// ---- POUs/Coolers/FB_SIM_RS_COMM_CRYOTELGT.TcPOU
FUNCTION_BLOCK FB_SIM_RS_COMM_CRYOTELGT EXTENDS FB_SIM_RS_COMM_BASE
VAR_INPUT
END_VAR
VAR_OUTPUT
END_VAR
VAR
	//
	// Status structure for Cryotel GT devices
	//
	// Status attributes that are read from the controller via RS-232
	sVersion:			STRING	:= 'v1.5.3 SIM';
	sMode:				STRING	:= 'GT';
	sSensor:			STRING	:= 'PT-100';
	sCtrlError:			STRING	:= '00000000';
	sCtrlMode:			STRING	:= 'OFF';
	
	lrPowerMeasured:	LREAL	:= 0.0;
	lrPowerCommanded:	LREAL	:= 240.0;
	lrTempColdHead:		LREAL	:= 289.15;	// Room temperature (289.15K = 16.0C) to start with.
	lrTempReject:		LREAL	:= 25.3;	// [C]
	lrTempTarget:		LREAL	:= 0.0;		// Not used
	
	
	fbTimer:		TON;

END_VAR

M_ActivityDo();	// Implement ramps, if any

SUPER^();

METHOD M_ActivityDo
VAR_INPUT
END_VAR
VAR
	lrProgress:	LREAL;
END_VAR
fbTimer();

IF sCtrlMode = 'POWER' THEN
	IF NOT fbTimer.Q	THEN
		lrProgress		:= TIME_TO_LREAL(fbTimer.ET) / TIME_TO_LREAL(fbTimer.PT);
		lrTempColdHead	:= 	289.15 - (289.15 - 80.0) * lrProgress;
	ELSE
		lrTempColdHead	:= 80.0;
	END_IF
END_IF
END_METHOD

METHOD M_GetSimReply : STRING(255)
VAR_INPUT
	{attribute 'OPC.UA.DA' := '0'}
	in_sReceived:	STRING(255);		// String received from a client
END_VAR
VAR
	sReply:	STRING(255);
	sTempStr:	STRING;
	lrVal:	LREAL;
	i:		INT;
    fbFormat   : FB_FormatString;
    sOut       : T_MaxString;
	nCh:	INT := 8;	// Number of channels for models 218 and 224
END_VAR
// Simulated reply has to include the echo of the command.
// For example:
//    command = 'VERSION'
//    reply   = 'VERSION$R$Nv1.5.3$R'

IF FIND (in_sReceived, 'VERSION') = 1 THEN
	sTempStr		:= CONCAT('VERSION$R$N', sVersion);
	M_GetSimReply	:= CONCAT(sTempStr,in_sReplySuffix);
ELSIF FIND (in_sReceived, 'MODE') = 1 THEN
	sTempStr		:= CONCAT('MODE$R$N', sMode);
	M_GetSimReply	:= CONCAT(sTempStr,in_sReplySuffix);
ELSIF FIND (in_sReceived, 'SENSOR') = 1 THEN
	sTempStr		:= CONCAT('SENSOR$R$N', sSensor);
	M_GetSimReply	:= CONCAT(sTempStr,in_sReplySuffix);
ELSIF FIND (in_sReceived, 'PWOUT=') = 1 THEN
	// Example:         'PWOUT=240$R'.
	// Reply should be: 'PWOUT=240$R$N240.00$R'.
	// Get the value from the command, i.e. everything after 'PWOUT='.
	sTempStr			:= MID(in_sReceived, LEN(in_sReceived)-6, 7);	// = '240$R'
	lrPowerCommanded	:= STRING_TO_LREAL(sTempStr);	// = 240.0
	sTempStr			:= CONCAT(in_sReceived, '$N');	// 'PWOUT=240$R' + '$N' = 'PWOUT=240$R$N' 
	M_GetSimReply		:= CONCAT(sTempStr, M_Get_LREAL_TO_STRING(lrPowerCommanded,2));
ELSIF FIND (in_sReceived, 'PWOUT') = 1 THEN
	M_GetSimReply	:= CONCAT('PWOUT$R$N', M_Get_LREAL_TO_STRING(lrPowerCommanded,2));
ELSIF FIND (in_sReceived, 'P') = 1 THEN
	lrPowerMeasured	:= M_GenerateRandom_LREAL(lrPowerCommanded-0.3,0.3);
	M_GetSimReply	:= CONCAT('P$R$N', M_Get_LREAL_TO_STRING(lrPowerMeasured,2));
ELSIF FIND (in_sReceived, 'ERROR') = 1 THEN
	sTempStr		:= CONCAT('ERROR$R$N', sCtrlError);
	M_GetSimReply	:= CONCAT(sTempStr,in_sReplySuffix);
ELSIF FIND (in_sReceived, 'COOLER=POWER') = 1 THEN
	sCtrlMode		:= 'POWER';
	M_GetSimReply	:= CONCAT('COOLER=POWER$R$NPOWER',in_sReplySuffix);
	// Start ramping down the cold head temperature,
	// starting fromroom temperature.
	lrTempColdHead	:= 289.15;	
	fbTimer(IN:=FALSE);
	fbTimer(IN:=TRUE, PT:=T#60S);
ELSIF FIND (in_sReceived, 'COOLER=OFF') = 1 THEN
	fbTimer(IN:=FALSE);	// Stop the temperature ramp.
	sCtrlMode			:= 'OFF';
	M_GetSimReply		:= CONCAT('COOLER=OFF$R$NOFF',in_sReplySuffix);
	lrPowerCommanded	:= 240.0;
	lrPowerMeasured		:= 0.0;
	lrTempColdHead		:= 289.15;
ELSIF FIND (in_sReceived, 'COOLER') = 1 THEN
	sTempStr		:= CONCAT('COOLER$R$N', sCtrlMode);
	M_GetSimReply	:= CONCAT(sTempStr,in_sReplySuffix);
ELSIF FIND (in_sReceived, 'TC') = 1 THEN
	M_GetSimReply	:= CONCAT('TC$R$N', M_Get_LREAL_TO_STRING(lrTempColdHead,2));
ELSIF FIND (in_sReceived, 'TEMP RJ') = 1 THEN
	// Reject temperature [C] !!! should always be close to 
	// the room temperature and slightly above the 
	// cold head temperature [K].
	// So, we have to convert K to C.
	lrTempReject	:= M_GenerateRandom_LREAL(MAX(16.0,lrTempColdHead-273.15),0.1);
	M_GetSimReply	:= CONCAT('TEMP RJ$R$N', M_Get_LREAL_TO_STRING(lrTempReject,2));
ELSE
	// Unknown command.
	// Return '<CR><LF><CR>', i.e. '$R$N$R' in order to complete the reading.
	M_GetSimReply	:= CONCAT('$R$N', in_sReplySuffix);
END_IF
END_METHOD

END_FUNCTION_BLOCK

// ---- POUs/Subsystems/Examples/Evacuation/FB_SIM_MICADO_VALVES.TcPOU
FUNCTION_BLOCK FB_SIM_MICADO_VALVES
VAR_INPUT
END_VAR
VAR_OUTPUT
END_VAR
VAR
	// Output valve control signals
	i_bON_PVV1	AT %I*:	BOOL;
	i_bON_PVV2	AT %I*:	BOOL;
	i_bON_PVV3	AT %I*:	BOOL;
	i_bON_PVV4	AT %I*:	BOOL;
	i_bON_GBV	AT %I*:	BOOL;
	
	
	// Simulation of ON/open feedback signal
	q_bON_PVV1	AT %Q*:	BOOL := FALSE;
	q_bON_PVV2	AT %Q*:	BOOL := FALSE;
	q_bON_PVV3	AT %Q*:	BOOL := FALSE;
	q_bON_PVV4	AT %Q*:	BOOL := FALSE;
	q_bON_GBV	AT %Q*:	BOOL := FALSE;
	
	// Simulation of OFF/closed feedback signal
	q_bOFF_PVV1	AT %Q*:	BOOL := TRUE;
	q_bOFF_PVV2	AT %Q*:	BOOL := TRUE;
	q_bOFF_PVV3	AT %Q*:	BOOL := TRUE;
	q_bOFF_PVV4	AT %Q*:	BOOL := TRUE;
	q_bOFF_GBV	AT %Q*:	BOOL := TRUE;
	

END_VAR

// ON signals are active low
q_bON_PVV1	:= i_bON_PVV1;
q_bON_PVV2	:= i_bON_PVV2;
q_bON_PVV3	:= i_bON_PVV3;
q_bON_PVV4	:= i_bON_PVV4;
q_bON_GBV	:= i_bON_GBV;


// OFF signals are active low
q_bOFF_PVV1	:= NOT i_bON_PVV1;
q_bOFF_PVV2	:= NOT i_bON_PVV2;
q_bOFF_PVV3	:= NOT i_bON_PVV3;
q_bOFF_PVV4	:= NOT i_bON_PVV4;
q_bOFF_GBV	:= NOT i_bON_GBV;

END_FUNCTION_BLOCK

// ---- POUs/Subsystems/Examples/Evacuation/FB_SIM_MICADO_PUMPS.TcPOU
FUNCTION_BLOCK FB_SIM_MICADO_PUMPS
VAR_INPUT
	in_RefPVP:	REFERENCE TO FB_CRYO_PUMP_ECODRY;
	in_RefTMP:	REFERENCE TO FB_CRYO_PUMP_ATH2303M;
	in_Delay:	TIME := T#10S;
END_VAR
VAR_OUTPUT
END_VAR
VAR
	trgStart_PVP:	R_TRIG;
	trgStart_TMP:	R_TRIG;
	trgStop_PVP:	F_TRIG;
	trgStop_TMP:	F_TRIG;
	
	timer_PVP:		TON;
	timer_TMP:		TON;
	
	bON_PVP:		BOOL := FALSE;
	bON_TMP:		BOOL := FALSE;
	
	q_PVP_Running	AT %Q*:	BOOL := TRUE;	// Active low!
	q_TMP_Ready		AT %Q*:	BOOL;
	q_TMP_Speed100	AT %Q*:	BOOL;
	
	ptrTMP_Speed:	POINTER TO DINT;
END_VAR

// Assign pointer to TMP speed.
ptrTMP_Speed	:= ADR(in_RefTMP.stat.nPumpSpeed);

// Get Start signals
trgStart_PVP(CLK:=in_RefPVP.in_bEnable);
trgStart_TMP(CLK:=in_RefTMP.in_bEnable);

// Get Stop signals
trgStop_PVP(CLK:=in_RefPVP.in_bEnable);
trgStop_TMP(CLK:=in_RefTMP.in_bEnable);

// Start timer on Start/Stop events
IF trgStart_PVP.Q THEN
	bON_PVP	:= TRUE;
	timer_PVP(IN:=FALSE);
	timer_PVP(IN:=TRUE, PT:=in_Delay/2);
ELSIF trgStop_PVP.Q THEN
	bON_PVP	:= FALSE;
	timer_PVP(IN:=FALSE);
	timer_PVP(IN:=TRUE, PT:=in_Delay/2);
END_IF

IF trgStart_TMP.Q THEN
	bON_TMP	:= TRUE;
	timer_TMP(IN:=FALSE);
	timer_TMP(IN:=TRUE, PT:=in_Delay);
ELSIF trgStop_TMP.Q THEN
	bON_TMP	:= FALSE;
	timer_TMP(IN:=FALSE);
	timer_TMP(IN:=TRUE, PT:=in_Delay * 2);
END_IF

// Execute timers
timer_PVP();
timer_TMP();

// Set outputs on timer expiry
IF timer_PVP.Q THEN
	// NOTE: PVP feedback is active low.
	IF bON_PVP THEN
		q_PVP_Running	:= FALSE;
	ELSE
		q_PVP_Running	:= TRUE;
	END_IF
END_IF

IF bON_TMP  AND (NOT timer_TMP.Q AND timer_TMP.ET > T#3S) THEN
	// Starting up.
	// Set speed > 100 rpm after 3 sec.
	ptrTMP_Speed^	:= 500;
	q_TMP_Speed100	:= TRUE;
END_IF

IF NOT bON_TMP  AND (NOT timer_TMP.Q AND timer_TMP.ET > T#5S) THEN
	// Stopping the pump.
	// Not ready after 5 sec.
	// However, the pump is still spinning.
	ptrTMP_Speed^	:= 1800;
	q_TMP_Ready		:= FALSE;
END_IF

IF timer_TMP.Q THEN
	IF bON_TMP THEN
		ptrTMP_Speed^	:= 2000;
		q_TMP_Ready	:= TRUE;
	ELSE
		ptrTMP_Speed^	:= 0;
		q_TMP_Ready		:= FALSE;
		q_TMP_Speed100	:= FALSE;
	END_IF
END_IF

END_FUNCTION_BLOCK

// ---- POUs/Subsystems/Examples/LN2_Precooling/FB_CRYO_LN2_PRECOOL.TcPOU
FUNCTION_BLOCK FB_CRYO_LN2_PRECOOL EXTENDS FB_CRYO_GEN_CTRL_BASE
VAR_INPUT
	in_lrTempK:				LREAL;			// Temperature input value [K]
	in_bTempValid:			BOOL := TRUE;	// Temperature Valid flag
	// Two parameters for decision making
	in_lrTempValveOpen:		LREAL := 91.27;		// Open  valve if temperature above this value [K]
	in_lrTempValveClose:	LREAL := 79.148;	// Close valve if temperature below this value [K]
END_VAR
VAR_OUTPUT
END_VAR
VAR
	// Status structure
	{attribute 'OPC.UA.DA' := '1'}
	stat:				T_CRYO_GEN_CTRL_STATUS_BASE;
	
	// LN2 valve
	valve:				FB_CRYO_VALVE_CTRL;
	bEnable_valve:		BOOL := FALSE;	// Valve open when bEnable_valve = TRUE
		

END_VAR

SUPER^();

METHOD M_ActionOffExecute
VAR_INPUT
END_VAR
//
// In this method the Enable flag of the valve is set to FALSE,
// meaning close the valve.
// 
// In the corresponding Activity M_ActivitySwitchingOff(), 
// the completion of the CLOSE/OFF command will be checked.
//
timer(IN:=FALSE);	// Reset Timer - mandatory!

// Close the valve
bEnable_valve	:= FALSE;
END_METHOD

METHOD M_ActionOnExecute
VAR_INPUT
END_VAR
//
// In this method the Enable flag of the valve is set to TRUE,
// meaning open the valve.
// 
// In the corresponding Activity M_ActivitySwitchingOn(), 
// the completion of the OPEN/ON command will be checked.
//
timer(IN:=FALSE);	// Reset Timer - mandatory!

// Close the valve
bEnable_valve	:= TRUE;
END_METHOD

METHOD M_ActivitySwitchingOff : BOOL
VAR_INPUT
END_VAR
//
// Wait for the valve to CLOSE/OFF.
// The valve state is available in its status structure.
// When complete, the method shall return TRUE, otherwise FALSE.


//
// Execute the timer - mandatory.
// Timer expiry is checked in M_ProcessEvents().
//
timer(IN:=TRUE, PT:=UDINT_TO_TIME(in_nTimeout));
	
// If valve is closed, return TRUE, otherwise FALSE.
IF valve.stat.bActOFF THEN
	M_ActivitySwitchingOff := TRUE;
ELSE
	M_ActivitySwitchingOff := FALSE;
END_IF
END_METHOD

METHOD M_ActivitySwitchingOn : BOOL
VAR_INPUT
END_VAR
//
// Wait for the valve to OPEN/ON.
// The valve state is available in its status structure.
// When complete, the method shall return TRUE, otherwise FALSE.


//
// Execute the timer - mandatory.
// Timer expiry is checked in M_ProcessEvents().
//
timer(IN:=TRUE, PT:=UDINT_TO_TIME(in_nTimeout));
	
// If valve is open, return TRUE, otherwise FALSE.
IF valve.stat.bActON THEN
	M_ActivitySwitchingOn := TRUE;
ELSE
	M_ActivitySwitchingOn := FALSE;
END_IF
END_METHOD

METHOD M_Configure
VAR_INPUT
END_VAR
// Configure the system and set the bConfigured flag to TRUE.

(*
	TODO USER: 
	- Set references to extended structures. e.g.
	     statRef REF=stat;
	- Configure the system.
*)

//	MUST be the very first line!!!
statRef REF=stat;

// The system has been configured
bConfigured := TRUE;
END_METHOD

METHOD M_ControlLoop : BOOL
VAR_INPUT
END_VAR
//
// This method implements the logic for controlling the LN2 valve.
// 
// The return value indicates if the valve should be OPEN/TRUE or CLOSED/FALSE
//
	
CASE statRef.nState OF
	E_CRYO_BIN_CTRL_STATE.ACTIVE_SWITCHING_ON,
	E_CRYO_BIN_CTRL_STATE.ACTIVE_ON:
		IF in_bTempValid AND in_lrTempK < in_lrTempValveClose THEN
			// Temperature too low.
			// Close the valve to stop cooling.
			M_ControlLoop	:= FALSE;
		ELSE
			// Keep the valve open
			M_ControlLoop	:= TRUE;
		END_IF

	E_CRYO_BIN_CTRL_STATE.ACTIVE_SWITCHING_OFF,
	E_CRYO_BIN_CTRL_STATE.ACTIVE_OFF:
		IF in_bTempValid AND in_lrTempK > in_lrTempValveOpen THEN
			// Temperature too high.
			// Open the valve to start cooling.
			M_ControlLoop	:= TRUE;
		ELSE
			// Keep the valve closed
			M_ControlLoop	:= FALSE;
		END_IF
ELSE
	// Keep the valve closed
	M_ControlLoop	:= FALSE;
END_CASE
END_METHOD

METHOD M_ExecuteActuators
VAR_INPUT
END_VAR
(*
	TODO USER: Execute all actuators, e.g. valve, heater, etc.
*)

valve(	in_nTimeout	:= 3000, 
		in_bEnable	:= bEnable_valve);
END_METHOD

METHOD M_IsError : BOOL
VAR_INPUT
END_VAR
//
// Check all possible failure conditions.
//
// This includes:
// - Configuration,
// - Validity of temperature reading,
// - Valve failure.
// 
// Return TRUE in case of errors.
// Set error description as well.
//
IF in_lrTempValveClose >= in_lrTempValveOpen THEN
	// The temperatue at which valve opens must be
	// higher than the one at which it closes.
	M_IsError	:= TRUE;
	stat.sError	:= 'ERROR: Wrong temperature limits!';
ELSIF NOT in_bTempValid	THEN
	// Temperature reading invalid.
	M_IsError	:= TRUE;
	stat.sError	:= 'ERROR: Reference temperature invalid!';
ELSIF valve.stat.bError 	THEN
	// Valve has failed.
	M_IsError	:= TRUE;
	stat.sError	:= 'ERROR: Valve failure!';
ELSE
	M_IsError	:= FALSE;
END_IF
END_METHOD

METHOD M_SetStatus
VAR_INPUT
END_VAR
// Execute M_SetStatus() of the base FB
SUPER^.M_SetStatus();


// Correct for LN2 specific labels

CASE statRef.nState OF
	
	E_CRYO_BIN_CTRL_STATE.ACTIVE_OFF:
	statRef.sState	:= 'ACTIVE_VALVE_CLOSED';
	
	E_CRYO_BIN_CTRL_STATE.ACTIVE_ON:
	statRef.sState	:= 'ACTIVE_VALVE_OPEN';
	
	E_CRYO_BIN_CTRL_STATE.ACTIVE_SWITCHING_ON:
	statRef.sState	:= 'OPENING VALVE...';
	
	E_CRYO_BIN_CTRL_STATE.ACTIVE_SWITCHING_OFF:
	statRef.sState	:= 'CLOSING VALVE...';
	
END_CASE
END_METHOD

END_FUNCTION_BLOCK

// ---- POUs/Actuators/FB_CRYO_GEN_CTRL_BASE.TcPOU
// Generic Controller
FUNCTION_BLOCK FB_CRYO_GEN_CTRL_BASE
VAR_INPUT
	in_bEnable:			BOOL := FALSE;	// Controller active while in_bEnable is TRUE
	in_nTimeout:		UDINT := 10000;	// Timeout for switching on/off [ms]. Default 10000.
	(*
		TODO USER: Add all specific input parameters, e.g.
		- Configuration parameters
		- External variables, e.g. temperature, pressure, etc.
	*)
END_VAR
VAR
	(*
		TODO USER: Add all system actuators, variables and I/O signals, e.g.
		
		{attribute 'OPC.UA.DA' := '1'}
		Actuator:	FB_CRYO_BIN_ACT;	// Heater, valve, etc.
	*)
	
	{attribute 'OPC.UA.DA' := '0'}
	statRef:	REFERENCE TO T_CRYO_GEN_CTRL_STATUS_BASE;

	(*
		TODO USER:	Add a 'stat' structure.
					It can be the T_CRYO_GEN_CTRL_STATUS or a struct that EXTENDS T_CRYO_GEN_CTRL_STATUS.
					For example:
						stat:	T_CRYO_BIN_CTRL_STATUS;
	*)
	
	nEvent:		E_CRYO_GEN_CTRL_EVENT := E_CRYO_GEN_CTRL_EVENT.NONE;

	{attribute 'OPC.UA.DA' := '0'}
	timer:		TON;		// Timer for commands
	
	{attribute 'OPC.UA.DA' := '0'}
	trgEnable:	R_TRIG;		// Rising trigger of in_bEnable
	
	// This flag will be set once M_Configure() is executed.
	bConfigured:	BOOL := FALSE;
END_VAR

// Don't do anything until the controller is configured
IF NOT bConfigured THEN
	M_Configure();
	RETURN;
END_IF

// Increment cycle counter
statRef.nCycleCounter := statRef.nCycleCounter + 1;



M_ReadInputs();


M_ExecuteActuators();


M_SetStatus();


M_CheckForEvents();


M_ProcessEvents();

METHOD M_ActionOffExecute
VAR_INPUT
END_VAR
//
// In this method the user shall turn off the actuator(s) such as valves, heaters, coolers, etc.
// Normally this is done by setting the in_bEnable flag of the actuator to FALSE.
// In the corresponding Activity M_ActivitySwitchingOff(), the completion of the OFF command shall be checked.
//
timer(IN:=FALSE);	// Reset Timer - mandatory!
END_METHOD

METHOD M_ActionOnExecute
VAR_INPUT
END_VAR
// In this method the user shall turn on the actuator(s) such as valves, heaters, coolers, etc.
// Normally this is done by setting the in_bEnable flag of the actuator to TRUE.
// In the corresponding Activity M_ActivitySwitchingOn(), the completion of the ON command shall be checked.
timer(IN:=FALSE);	// Reset Timer
END_METHOD

METHOD M_ActivitySwitchingOff : BOOL
VAR_INPUT
END_VAR
// In this method the user shall wait until the actuator is turned OFF.
// The actuator state is available in the status structure.
// When complete, the method shall return TRUE, otherwise FALSE.


// Dummy implementation.
// Complete after 5 sec.
//
timer(IN:=TRUE, PT:=UDINT_TO_TIME(in_nTimeout));
	
IF timer.ET >= T#5S THEN
	M_ActivitySwitchingOff := TRUE;
ELSE
	M_ActivitySwitchingOff := FALSE;
END_IF
END_METHOD

METHOD M_ActivitySwitchingOn : BOOL
VAR_INPUT
END_VAR
// In this method the user shall wait until the actuator is turned ON.
// The actuator state is available in the status structure.
// When complete, the method shall return TRUE, otherwise FALSE.


// Dummy implementation.
// Complete after 5 sec.
//
timer(IN:=TRUE, PT:=UDINT_TO_TIME(in_nTimeout));
	
IF timer.ET >= T#5S THEN
	M_ActivitySwitchingOn := TRUE;
ELSE
	M_ActivitySwitchingOn := FALSE;
END_IF
END_METHOD

METHOD M_CheckForEvents
VAR_INPUT
END_VAR
VAR
	nEventTmp:	E_CRYO_GEN_CTRL_EVENT := E_CRYO_GEN_CTRL_EVENT.NONE;
END_VAR
// TODO USER
//

nEventTmp	:= E_CRYO_GEN_CTRL_EVENT.NONE;

// Check for the Enable trigger
trgEnable(CLK := in_bEnable);


CASE statRef.nState OF
	/////////////////////////////////
	E_CRYO_BIN_CTRL_STATE.NONE:
	/////////////////////////////////
	//
	// This is the state on power-up.
	statRef.nState	:= E_CRYO_BIN_CTRL_STATE.OFF;
	

	/////////////////////////////////
	E_CRYO_BIN_CTRL_STATE.OFF:
	/////////////////////////////////
	//
	IF	trgEnable.Q  THEN
		nEventTmp	:= E_CRYO_GEN_CTRL_EVENT.ENABLE;
	END_IF
	
	
	/////////////////////////////////
	E_CRYO_BIN_CTRL_STATE.ACTIVE_OFF:
	/////////////////////////////////
	//
	IF NOT in_bEnable  THEN
		// Goto Off.
		//
		nEventTmp	:= E_CRYO_GEN_CTRL_EVENT.DISABLE;
	ELSIF M_ControlLoop() = TRUE THEN
		nEventTmp	:= E_CRYO_GEN_CTRL_EVENT.ON;
	END_IF
	
	
	//////////////////////////////////////////
	E_CRYO_BIN_CTRL_STATE.ACTIVE_SWITCHING_ON:
	//////////////////////////////////////////
	//
	IF NOT in_bEnable  THEN
		// Goto ACTIVE_OF first.
		//
		nEventTmp	:= E_CRYO_GEN_CTRL_EVENT.OFF;
	ELSIF timer.Q THEN
		nEventTmp	:= E_CRYO_GEN_CTRL_EVENT.ERROR;
	ELSIF M_ControlLoop() = FALSE THEN
		nEventTmp	:= E_CRYO_GEN_CTRL_EVENT.OFF;
	ELSIF M_ActivitySwitchingOn() THEN
		nEventTmp	:= E_CRYO_GEN_CTRL_EVENT.IS_ON;
	END_IF
	

	//////////////////////////////////////////
	E_CRYO_BIN_CTRL_STATE.ACTIVE_ON:
	//////////////////////////////////////////
	//
	IF NOT in_bEnable  THEN
		// Goto ACTIVE_OFF first.
		//
		nEventTmp	:= E_CRYO_GEN_CTRL_EVENT.OFF;
	ELSIF M_ControlLoop() = FALSE THEN
		nEventTmp	:= E_CRYO_GEN_CTRL_EVENT.OFF;
	END_IF
	

	///////////////////////////////////////////
	E_CRYO_BIN_CTRL_STATE.ACTIVE_SWITCHING_OFF:
	///////////////////////////////////////////
	//
	IF NOT in_bEnable  THEN
		// Goto Off.
		//
		nEventTmp	:= E_CRYO_GEN_CTRL_EVENT.DISABLE;
	ELSIF timer.Q THEN
		nEventTmp	:= E_CRYO_GEN_CTRL_EVENT.ERROR;
	ELSIF M_ControlLoop() = TRUE THEN
		nEventTmp	:= E_CRYO_GEN_CTRL_EVENT.ON;
	ELSIF M_ActivitySwitchingOff() THEN
		nEventTmp	:= E_CRYO_GEN_CTRL_EVENT.IS_OFF;
	END_IF
	

	/////////////////////////////////
	E_CRYO_BIN_CTRL_STATE.ERROR:
	/////////////////////////////////
	//
	IF	trgEnable.Q  THEN
		nEventTmp	:= E_CRYO_GEN_CTRL_EVENT.ENABLE;
	END_IF
	
END_CASE

nEvent	:= nEventTmp;
END_METHOD

METHOD M_Configure
VAR_INPUT
END_VAR
// Configure the system and set the bConfigured flag to TRUE.

(*
	TODO USER: 
	- Set references to extended structures. e.g.
	- Configure the system, if any.
	
	MUST be the very first line!!!
	     statRef REF=stat;
*)

// The system has been configured
bConfigured := TRUE;
END_METHOD

METHOD M_ControlLoop : BOOL
VAR_INPUT
END_VAR
VAR_INST
	timerDummy:	TON;	// Dummy timer
	nDummy:		UDINT;	// Dummy counter
END_VAR
// Dummy implementation of the control loop.
// The return value says if the loop should be ACTIVE/TRUE or INACTIVE/FALSE

IF nDummy = 0 THEN
	timerDummy(IN:=FALSE);	// Reset timer
END_IF
nDummy	:= nDummy + 1;

timerDummy(IN:=TRUE, PT:=T#10S);

CASE statRef.nState OF
	E_CRYO_BIN_CTRL_STATE.ACTIVE_SWITCHING_OFF,
	E_CRYO_BIN_CTRL_STATE.ACTIVE_OFF:
		IF timerDummy.Q THEN
			nDummy := 0;
			// This will create ON event.
			M_ControlLoop	:= TRUE;
		ELSE
			// Remain OFF
			M_ControlLoop	:= FALSE;
		END_IF
	E_CRYO_BIN_CTRL_STATE.ACTIVE_SWITCHING_ON,
	E_CRYO_BIN_CTRL_STATE.ACTIVE_ON:
		IF timerDummy.Q THEN
			nDummy := 0;
			// This will create OFF event.
			M_ControlLoop	:= FALSE;
		ELSE
			// Remain ON
			M_ControlLoop	:= TRUE;
		END_IF
	ELSE
		M_ControlLoop	:= FALSE;
END_CASE
END_METHOD

METHOD M_ExecuteActuators
VAR_INPUT
END_VAR
(*
	TODO USER: Execute all actuators, e.g. valve, heater, etc.


// Example: Execute Actuator FB instance
Actuator(
	in_nFeedback		:= in_nFeedback,
	in_nTimeout			:= in_nTimeout,
	in_bActiveLowCtrl	:= in_bActiveLowCtrl,
	in_bActiveLowStat	:= in_bActiveLowStat);


*)
END_METHOD

METHOD M_IsError : BOOL
VAR_INPUT
END_VAR
(*
	TODO USER: Do all the checks and return TRUE if error.
	Otherwise, return FALSE (no error).
*)

M_IsError	:= FALSE;
END_METHOD

METHOD M_ProcessEvents
VAR_INPUT
END_VAR
// TODO USER
//


CASE statRef.nState OF
	/////////////////////////////////
	E_CRYO_BIN_CTRL_STATE.NONE:
	/////////////////////////////////
	//
	// Nothing to do.
	;
	

	/////////////////////////////////
	E_CRYO_BIN_CTRL_STATE.OFF:
	/////////////////////////////////
	//
	IF	nEvent = E_CRYO_GEN_CTRL_EVENT.ENABLE  THEN
		// Activate the control loop.
		// Goto Active_Off first.
		//
		M_ActionOffExecute();		
		// Set next state
		statRef.nState	:= E_CRYO_BIN_CTRL_STATE.ACTIVE_SWITCHING_OFF;
	END_IF
	
	
	/////////////////////////////////
	E_CRYO_BIN_CTRL_STATE.ACTIVE_OFF:
	/////////////////////////////////
	//
	IF	nEvent = E_CRYO_GEN_CTRL_EVENT.DISABLE  THEN
		// Goto Off.
		//
		// Set next state
		statRef.nState	:= E_CRYO_BIN_CTRL_STATE.OFF;
	ELSIF nEvent = E_CRYO_GEN_CTRL_EVENT.ON THEN
		M_ActionOnExecute();
		// Set next state
		statRef.nState	:= E_CRYO_BIN_CTRL_STATE.ACTIVE_SWITCHING_ON;
	END_IF
	
	
	//////////////////////////////////////////
	E_CRYO_BIN_CTRL_STATE.ACTIVE_SWITCHING_ON:
	//////////////////////////////////////////
	//
	// Check for timeout
	IF timer.Q THEN
		// Goto ERROR state
		statRef.nState	:= E_CRYO_BIN_CTRL_STATE.ERROR;
	ELSIF nEvent = E_CRYO_GEN_CTRL_EVENT.OFF THEN
		M_ActionOffExecute();
		// Set next state
		statRef.nState	:= E_CRYO_BIN_CTRL_STATE.ACTIVE_SWITCHING_OFF;
	ELSIF M_ActivitySwitchingOn() THEN
		statRef.nState	:= E_CRYO_BIN_CTRL_STATE.ACTIVE_ON;
	END_IF
	

	/////////////////////////////////
	E_CRYO_BIN_CTRL_STATE.ACTIVE_ON:
	/////////////////////////////////
	//
	IF	nEvent = E_CRYO_GEN_CTRL_EVENT.DISABLE  THEN
		// Goto Off.
		//
		M_ActionOffExecute();
		// Set next state
		statRef.nState	:= E_CRYO_BIN_CTRL_STATE.ACTIVE_SWITCHING_OFF;
	ELSIF nEvent = E_CRYO_GEN_CTRL_EVENT.OFF THEN
		M_ActionOffExecute();
		// Set next state
		statRef.nState	:= E_CRYO_BIN_CTRL_STATE.ACTIVE_SWITCHING_OFF;
	END_IF
	
	
	///////////////////////////////////////////
	E_CRYO_BIN_CTRL_STATE.ACTIVE_SWITCHING_OFF:
	///////////////////////////////////////////
	//
	// Check for timeout
	IF timer.Q THEN
		// Goto ERROR state
		statRef.nState	:= E_CRYO_BIN_CTRL_STATE.ERROR;
	ELSIF nEvent = E_CRYO_GEN_CTRL_EVENT.ON THEN
		M_ActionOnExecute();
		// Set next state
		statRef.nState	:= E_CRYO_BIN_CTRL_STATE.ACTIVE_SWITCHING_ON;
	ELSIF M_ActivitySwitchingOff() THEN
		statRef.nState	:= E_CRYO_BIN_CTRL_STATE.ACTIVE_OFF;
	END_IF

	
	/////////////////////////////////
	E_CRYO_BIN_CTRL_STATE.ERROR:
	/////////////////////////////////
	//
	IF	nEvent = E_CRYO_GEN_CTRL_EVENT.ENABLE  THEN
		// Activate the control loop.
		// Goto Active_Off first.
		//
		// Set next state
		statRef.nState	:= E_CRYO_BIN_CTRL_STATE.ACTIVE_OFF;
	END_IF
	
END_CASE


// If error, goto ERROR state.
IF M_IsError() THEN
	statRef.nState	:= E_CRYO_BIN_CTRL_STATE.ERROR;
END_IF

// Set status
M_SetStatus();
END_METHOD

METHOD M_ReadInputs
VAR_INPUT
END_VAR
(*
	TODO USER: Read all inputs and assign values to variables.
	Inputs can be pressure, temperature, etc.
*)
END_METHOD

METHOD M_SetStatus
VAR_INPUT
END_VAR
CASE statRef.nState OF
	
	E_CRYO_BIN_CTRL_STATE.OFF:
	statRef.bDone	:= TRUE;
	statRef.bBusy	:= FALSE;
	statRef.bError	:= FALSE;
	statRef.bActive	:= FALSE;
	statRef.sState	:= 'OFF';
	
	E_CRYO_BIN_CTRL_STATE.ACTIVE_OFF:
	statRef.bDone	:= TRUE;
	statRef.bBusy	:= FALSE;
	statRef.bError	:= FALSE;
	statRef.bActive	:= TRUE;
	statRef.sState	:= 'ACTIVE_OFF';
	
	E_CRYO_BIN_CTRL_STATE.ACTIVE_ON:
	statRef.bDone	:= TRUE;
	statRef.bBusy	:= FALSE;
	statRef.bError	:= FALSE;
	statRef.bActive	:= TRUE;
	statRef.sState	:= 'ACTIVE_ON';
	
	E_CRYO_BIN_CTRL_STATE.ACTIVE_SWITCHING_ON:
	statRef.bDone	:= FALSE;
	statRef.bBusy	:= TRUE;
	statRef.bError	:= FALSE;
	statRef.bActive	:= TRUE;
	statRef.sState	:= 'ACTIVE_SWITCHING_ON...';
	
	E_CRYO_BIN_CTRL_STATE.ACTIVE_SWITCHING_OFF:
	statRef.bDone	:= FALSE;
	statRef.bBusy	:= TRUE;
	statRef.bError	:= FALSE;
	statRef.bActive	:= TRUE;
	statRef.sState	:= 'ACTIVE_SWITCHING_OFF...';
	
	E_CRYO_BIN_CTRL_STATE.ERROR:
	statRef.bDone	:= TRUE;
	statRef.bBusy	:= FALSE;
	statRef.bError	:= TRUE;
	statRef.bActive	:= FALSE;
	statRef.sState	:= 'ERROR';

END_CASE

IF NOT statRef.bError THEN
	statRef.sError := 'OK';
END_IF
END_METHOD

END_FUNCTION_BLOCK

// ---- POUs/Subsystems/Examples/LN2_Precooling/FB_SIM_LN2_PRECOOL.TcPOU
FUNCTION_BLOCK FB_SIM_LN2_PRECOOL
VAR_INPUT
	ln2Ref:	REFERENCE TO FB_CRYO_LN2_PRECOOL;
END_VAR
VAR_OUTPUT
	lrTempK:	LREAL;	// Simulated temperature value [K]
END_VAR
VAR
	SIM_ln2_temp:	FB_CRYO_SIM_TEMPERATURE;	// Simulated temperature FB
	
	trgEnable:		R_TRIG;						// Precooling  enable change trigger
	trgDisable:		F_TRIG;						// Precooling disable change trigger
	trgState:		R_TRIG;						// State change trigger

	nState:			E_CRYO_BIN_CTRL_STATE	:= E_CRYO_BIN_CTRL_STATE.NONE;
	
END_VAR

// Detect change of LN2 system Enable 
trgEnable(CLK := ln2Ref.in_bEnable);

// Detect change of LN2 system Disable 
trgDisable(CLK := ln2Ref.in_bEnable);

// Detect change of LN2 system State 
trgState(CLK := (	(ln2Ref.stat.nState = E_CRYO_BIN_CTRL_STATE.ACTIVE_ON OR 
					 ln2Ref.stat.nState = E_CRYO_BIN_CTRL_STATE.ACTIVE_OFF) 	AND 
					ln2Ref.stat.nState <> nState));

IF trgEnable.Q	THEN
	// System enabled.

	// Save current state
	nState	:= ln2Ref.stat.nState;
	
	// Start changing temperature just to get the system 
	// working for the first time.
	IF SIM_ln2_temp.lrTempK >= ln2Ref.in_lrTempValveClose	THEN
		// Lower simulated temperature to lower limit -1 deg in 5 sec.
		SIM_ln2_temp.M_RampTo(ln2Ref.in_lrTempValveClose - 1, 5000);
	ELSE
		// Rise simulated temperature to upper limit +1 deg in 5 sec.
		SIM_ln2_temp.M_RampTo(ln2Ref.in_lrTempValveOpen + 1, 5000);
	END_IF
ELSIF trgDisable.Q	THEN
	// System disabled. Stop the temperature ramp.
	SIM_ln2_temp.M_Stop();	
ELSIF ln2Ref.in_bEnable AND trgState.Q	THEN
	// State of enabled system changed.
	// Save new state
	nState	:= ln2Ref.stat.nState;
	
	// Start a ramp, depending on the new state.
	IF ln2Ref.stat.nState = E_CRYO_BIN_CTRL_STATE.ACTIVE_ON	THEN
		// Valve open, the temperature should start falling.
		// Ramp it down to the CLOSE limit minus 1 deg in 10 sec.
		SIM_ln2_temp.M_RampTo(ln2Ref.in_lrTempValveClose - 1.0, 10000);
	ELSIF ln2Ref.stat.nState = E_CRYO_BIN_CTRL_STATE.ACTIVE_OFF	THEN
		// Valve closed, the temperature should start rising.
		// Ramp it up to the OPEN limit plus 1 deg in 10 sec.
		SIM_ln2_temp.M_RampTo(ln2Ref.in_lrTempValveOpen + 1.0, 10000);
	END_IF
END_IF


// Execute temperature simulator FB.
SIM_ln2_temp();

// Assign the simulated temperature to the output var
lrTempK	:= SIM_ln2_temp.lrTempK;

END_FUNCTION_BLOCK

// ---- POUs/Sensors/FB_CRYO_SBG232.TcPOU
FUNCTION_BLOCK FB_CRYO_SBG232
VAR_INPUT
	in_sName:		string	   := 'IO-Link SBG232';
	in_sUnitFlow:	STRING(16) := 'L/min';	//	Units for Flow, default [L/min] 
	in_sUnitTemp:	STRING(16) := '°C';		//	Units for Temperature, default [°C] 
END_VAR
VAR_OUTPUT
END_VAR
VAR
	//
	// Variables to be linked
	//
	
	// InfoData -> State of IO-Link master, e.g. EL6224.
	i_nCouplerState			AT %I*:	UINT;	
	// DeviceState Inputs -> State Ch# of IO-Link master, e.g. EL6224.
	i_nDeviceStateInputCh	AT %I*:	USINT;	
	// Raw device data: IO-Link Port# -> Port#:process data
	i_ArrPortProcessData	AT %I*:	ARRAY [0..3] OF USINT;
	
	
	stat:	T_CRYO_SBG232_STAT;
	
END_VAR

// Configure if it hasn't been done.
M_Configure();

// Extract sensor reading from the raw value.
M_UpdateStatus();

METHOD M_Configure
VAR_INPUT
END_VAR
IF NOT stat.bConfigured	THEN
	stat.bConfigured	:= TRUE;
	
	stat.sName			:= in_sName;
	
	stat.flow.sUnits	:= in_sUnitFlow;
	stat.temp.sUnits	:= in_sUnitTemp;

	stat.flow.sType		:= 'Flow';
	stat.temp.sType		:= 'Temperature';

END_IF
END_METHOD

METHOD M_SetError
VAR_INPUT
	nSensor:	E_CRYO_SBG232_SENSOR_TYPE;
	sError:		STRING;
END_VAR
VAR
	refSensor:	REFERENCE TO T_CRYO_IOLINK_SENSOR_STATUS;
END_VAR
IF nSensor	= E_CRYO_SBG232_SENSOR_TYPE.FLOW	THEN
	refSensor	REF=stat.flow;
ELSIF nSensor	= E_CRYO_SBG232_SENSOR_TYPE.TEMP	THEN
	refSensor	REF=stat.temp;
END_IF

refSensor.bError		:= TRUE;
refSensor.bInRange		:= FALSE;
refSensor.bValid		:= FALSE;
refSensor.sStatus		:= sError;
END_METHOD

METHOD M_SetReading
VAR_INPUT
	nSensor:	E_CRYO_SBG232_SENSOR_TYPE;
	lrValue:	LREAL;
END_VAR
VAR
	refSensor:	REFERENCE TO T_CRYO_IOLINK_SENSOR_STATUS;
END_VAR
IF nSensor	= E_CRYO_SBG232_SENSOR_TYPE.FLOW	THEN
	refSensor	REF=stat.flow;
ELSIF nSensor	= E_CRYO_SBG232_SENSOR_TYPE.TEMP	THEN
	refSensor	REF=stat.temp;
END_IF

refSensor.bOverrange	:= FALSE;
refSensor.bUnderrange	:= FALSE;
refSensor.bError		:= FALSE;
refSensor.bInRange		:= TRUE;
refSensor.bValid		:= TRUE;
refSensor.lrValue		:= lrValue;
refSensor.sStatus		:= 'OK';
END_METHOD

METHOD M_UpdateStatus
VAR_INPUT
END_VAR
VAR
	lrVal:	LREAL;
END_VAR
// General check if the EL6224 and IO-Link are OK.
IF i_nCouplerState	<> 8	THEN
	stat.sStatus	:= 'IO-Link terminal not in OP state. Check the mapping.';
	M_SetError(E_CRYO_SBG232_SENSOR_TYPE.FLOW, 'IO-Link terminal not in OP state');
	M_SetError(E_CRYO_SBG232_SENSOR_TYPE.TEMP, 'IO-Link terminal not in OP state');
	RETURN;
ELSIF i_nDeviceStateInputCh	<> 3	THEN
	stat.sStatus	:= 'IO-Link Channel not in OP state';
	M_SetError(E_CRYO_SBG232_SENSOR_TYPE.FLOW, 'IO-Link Channel not in OP state');
	M_SetError(E_CRYO_SBG232_SENSOR_TYPE.TEMP, 'IO-Link Channel not in OP state');
	RETURN;
ELSE
	stat.sStatus	:= 'OK';
END_IF


//////////////
// Flow
//////////////

lrVal	:= (256.0 * i_ArrPortProcessData[0] + i_ArrPortProcessData[1]) / 100.0;
stat.flow.lrValue	:= lrVal;

IF lrVal = 18.05	THEN
	stat.flow.bOverrange	:= TRUE;
	stat.flow.bUnderrange	:= FALSE;
	M_SetError(E_CRYO_SBG232_SENSOR_TYPE.FLOW, 'Overrange');
ELSE
	M_SetReading(E_CRYO_SBG232_SENSOR_TYPE.FLOW, lrVal);
END_IF


////////////////
// Temperature
////////////////

lrVal	:= TRUNC(256.0 * i_ArrPortProcessData[2] + i_ArrPortProcessData[3]) / 4;	// /4 = SHR(2)
stat.temp.lrValue	:= lrVal;


IF lrVal = 123.0	THEN
	stat.temp.bOverrange	:= TRUE;
	stat.temp.bUnderrange	:= FALSE;
	M_SetError(E_CRYO_SBG232_SENSOR_TYPE.TEMP, 'Overrange');
ELSIF lrVal = -33.0	THEN
	stat.temp.bOverrange	:= FALSE;
	stat.temp.bUnderrange	:= TRUE;
	M_SetError(E_CRYO_SBG232_SENSOR_TYPE.TEMP, 'Underrange');
ELSE
	M_SetReading(E_CRYO_SBG232_SENSOR_TYPE.TEMP, lrVal);
END_IF
END_METHOD

END_FUNCTION_BLOCK

// ---- POUs/Simulation/FB_CRYO_SIM_SBG232.TcPOU
FUNCTION_BLOCK FB_CRYO_SIM_SBG232
VAR_INPUT
	in_lrRefTemp:	LREAL := 21.0;	// Temperature reference point [°C]
	in_lrRefFlow:	LREAL := 4.30;	// Flow reference point [L/min]
	in_lrVarTemp:	LREAL := 2.0;	// Temperature reading variation [°C]
	in_lrVarFlow:	LREAL := 0.1;	// Flow reading variation [L/min]
END_VAR
VAR_OUTPUT
END_VAR
VAR
	temp:	FB_CRYO_SIM_SINE;	// Temperature variation as sine wave
	flow:	FB_CRYO_SIM_SINE;	// Flow variation as sine wave
	
	lrTemp:	LREAL;
	lrFlow:	LREAL;
	nWord:	WORD;
	
	q_nCouplerState			AT %Q*:	UINT	:= 8;
	q_nDeviceStateInputCh	AT %Q*:	USINT	:= 3;
	q_ArrPortProcessData	AT %Q*:	ARRAY [0..3] OF BYTE;
END_VAR

// Simulate temperature and flow variations as sinewaves
temp(in_lrAmplitude:=in_lrVarTemp, in_nPeriod:=60000);
flow(in_lrAmplitude:=in_lrVarFlow, in_nPeriod:=120000);

// Calculate simulated values
lrTemp	:= in_lrRefTemp + temp.out_lrValue;
lrFlow	:= in_lrRefFlow + flow.out_lrValue;


// Set output variables

////////////////
// Temperature
////////////////

// lrVal	:= TRUNC(256.0 * i_ArrPortProcessData[2] + i_ArrPortProcessData[3]) / 4;	// /4 = SHR(2)
nWord	:= LREAL_TO_WORD(lrTemp	* 4);
q_ArrPortProcessData[2]	:= UINT_TO_BYTE(16#FF AND SHR(nWord,8));
q_ArrPortProcessData[3]	:= UINT_TO_BYTE(16#FF AND nWord);


//////////////
// Flow
//////////////

// lrVal	:= (256.0 * i_ArrPortProcessData[0] + i_ArrPortProcessData[1]) / 100.0;
nWord	:= LREAL_TO_WORD(lrFlow	* 100.0);
q_ArrPortProcessData[0]	:= UINT_TO_BYTE(16#FF AND SHR(nWord,8));
q_ArrPortProcessData[1]	:= UINT_TO_BYTE(16#FF AND nWord);

END_FUNCTION_BLOCK

// ---- GlobalTextList.TcGTLO
TEXTLIST GlobalTextList
  890 = ''
  626 = '\nCCC'
  727 = '\nHeater'
  810 = '\n\nBench'
  769 = '\n\nCCC'
  26 = '\nBench'
  726 = '\nDetector'
  935 = '\nHeater'
  730 = '         Detector'
  245 = '%.02f'
  143 = '%.03f'
  939 = '%.0f'
  303 = '%.1e'
  876 = '%.1f'
  556 = '%.1f '
  219 = '%.1f %'
  321 = '%.1f %%'
  723 = '%.1f C'
  310 = '%.1f K'
  495 = '%.1f K/min'
  74 = '%.2e'
  454 = '%.2e mbar'
  622 = '%.2f'
  844 = '%.2f A'
  706 = '%.2f K'
  254 = '%.3e'
  1040 = '%.3e mbar'
  306 = '%.3f K'
  686 = '%0.3f'
  778 = '%d'
  241 = '%d rpm'
  154 = '%s'
  996 = '%u'
  330 = "'COOLER' command: Cooler Control Mode: OFF or POWER"
  842 = "'MODE' command: Cryocooler type, e.g. GT"
  539 = "'P' command: Measured Power"
  533 = "'PWOUT' command: Commanded power"
  736 = "'SENSOR' command: Configured temp. sensor type, e.g. 'PT-100'"
  381 = "'Simulated value [K] when simulation is active.'"
  536 = "'TC' command: Cold Head temperature"
  540 = "'TEMP RJ' command: Reject Temperature"
  546 = "'TTARGET' command: TargetTemperature"
  2300 = "'Value used by the system [C]'"
  94 = "'Value used by the system [K]'"
  155 = "'VERSION' command: Current controller code version"
  995 = "'°C'"
  1875 = "'°K'"
  407 = '-'
  44 = '0x%04X'
  553 = '1.0 K/min'
  138 = '100'
  248 = '100.0 %'
  299 = '273.15 K'
  653 = '273.15 K %'
  997 = 'Activate Simulation'
  331 = 'Active   ON     Error'
  790 = 'Actual             Threshold'
  1017 = 'Actual Cmd'
  1932 = 'Actual command going out'
  2155 = 'Actual Simulation flag'
  2686 = 'Actual Simulation flag going out'
  1586 = 'Actual Simulation flag set the user'
  1303 = 'Actual Valve command '
  746 = 'Alarm :'
  240 = 'Ambient'
  757 = 'At Speed [%] :'
  849 = 'AUTO'
  1295 = 'AUTO Cmd'
  6 = 'AUTO Simulation flag'
  1861 = 'AUTO Simulation flag set by the system'
  427 = 'Bearing Counter [%] :'
  1470 = 'Bearing Warning [%] :'
  32 = 'Bench'
  256 = 'C'
  548 = 'CCC'
  144 = 'CCC Control is Enabled/Active'
  329 = 'CCC is ON'
  1058 = 'CLOSE'
  786 = 'Cold Head [K] :'
  872 = 'Coldest Point'
  183 = 'Coldest point in the Cryostat'
  216 = 'Command coming from the Control System'
  994 = 'Commanded [W] :'
  523 = 'Compressor Year: '
  640 = 'Configuration'
  317 = 'Control'
  284 = 'Control Mode'
  821 = 'Controllers'
  328 = 'COOL'
  462 = 'Cooler State'
  532 = 'Cryo Controller'
  637 = 'Cryo pressure [mbar]'
  146 = 'Cryostat Pressure [mbar]:'
  439 = 'Ctrl Signal :'
  989 = 'Current: '
  1206 = 'Deactivate Simulation'
  600 = 'deg C'
  304 = 'deg K'
  788 = 'Delta Pressure\n%4.1f bar'
  925 = 'DET - Coldest'
  466 = 'DET-Coldest'
  316 = 'Detector'
  784 = 'Drive Elec. Hours :'
  133 = 'Drive Elec. Temp [°C] :'
  49 = 'Drive Status'
  308 = 'Electronics Drive Temp.'
  235 = 'EMCY Closed'
  806 = 'ENABLE'
  998 = 'Enable'
  1445 = 'ENG'
  1572 = 'Engineering / Commissioning Mode'
  238 = 'Error'
  905 = 'Error :'
  280 = 'Error description'
  325 = 'Error Status'
  700 = 'Evac'
  234 = 'Evac Valve'
  205 = 'EVACUATE'
  230 = 'Evacuate'
  692 = 'Evacuation System'
  258 = 'Evacuation System Status'
  67 = 'Exhaust'
  96 = 'Flag if Heater RAMP is On'
  25 = 'Flag if reading is in sensor range'
  688 = 'Frequency Reference'
  837 = 'FW Version'
  1833 = 'FW Version :'
  1216 = 'GBV'
  315 = 'GUI'
  54 = 'Heat Shield Temperature'
  724 = 'Heater'
  829 = 'Heater Control is Enabled/Active'
  856 = 'Heater is ON'
  642 = 'Heater Output [%]'
  447 = 'Heater Ramp Rate'
  202 = 'Heater Range'
  543 = 'Helium\n%4.1f ºC'
  909 = 'High Pressure\n%4.1f bar'
  474 = 'Hours: '
  830 = 'HTR'
  858 = 'HW Version'
  2127 = 'HW Version :'
  51 = 'Hz'
  873 = 'ID'
  218 = 'If active, system is enabled'
  628 = 'If ON, compressor is running'
  5 = 'If ON, compressor is simulated'
  145 = 'If ON, control output signal is active.'
  731 = 'If ON, Cooler is simulated.'
  1779 = 'If ON, ENG command is not safe!'
  878 = 'If ON, Evacuation System is in ERROR state.'
  159 = 'If ON, Insulation Valve is OPEN'
  389 = 'If ON, Pump is Running'
  111 = 'If ON, reading is in error.'
  1927 = 'If ON, reading is in expected range.'
  70 = 'If ON, reading is in overrange.'
  1941 = 'If ON, reading is in underrange.'
  869 = 'If ON, reading is valid.'
  949 = 'If ON, system is enabled'
  9 = 'If ON, system is in ERROR state.'
  942 = 'If ON, there is a communication problem with the Cooler.'
  2000 = 'If ON, there is an error in the SW implementation of permission handling.'
  1062 = 'If ON, there was an error'
  182 = 'If ON, TMP pump is at its nominal speed, i.e. Ready.'
  561 = 'If ON, TMP pump is still spinning.'
  112 = 'In Range'
  233 = 'In Vacuum'
  687 = 'Inlet'
  47 = 'Input Terminal Status'
  659 = 'INTERLOCK'
  1474 = 'Interlock'
  475 = 'IRATEC Cryo Controller'
  2484 = 'K'
  406 = 'kW'
  717 = 'Lakeshore'
  242 = 'LN2'
  322 = 'LN2 OFF'
  33 = 'LN2 Pre-Cooling'
  106 = 'Low Pressure\n%4.1f bar'
  285 = 'mA'
  98 = 'MANUAL'
  172 = 'mbar'
  347 = 'Measured [W] :'
  395 = 'Mirror'
  336 = 'Motor Current'
  257 = 'Motor Current [mA] :'
  157 = 'Motor Power [W] :'
  698 = 'Motor Voltage'
  804 = 'Motor Voltage [V] :'
  27 = 'NO-SIM'
  396 = 'Nominal Speed [rpm] :'
  708 = 'OFF'
  518 = 'Oil\n%4.1f ºC'
  611 = 'OK for Process, i.e. speed ≥ nominal speed'
  1093 = 'ON'
  229 = 'Open'
  1381 = 'OPEN'
  791 = 'Operational State'
  1080 = 'OUTPUT Cmd'
  689 = 'Output Frequency'
  46 = 'Output Power'
  48 = 'Output Terminal Status'
  691 = 'Output Voltage Reference'
  1982 = 'Overrange'
  1437 = 'Permit CLOSE'
  803 = 'Permit OFF'
  93 = 'Permit ON'
  1308 = 'Permit OPEN'
  239 = 'PID'
  732 = 'Power'
  403 = 'PRE COOL'
  598 = 'PRE-COOL'
  586 = 'PRECOOL'
  413 = 'presence of a warning'
  636 = 'presence of an alarm'
  705 = 'Pressure threshold for safe opening of the pre-vacuum valve [mbar]'
  1182 = 'Pressure threshold for safe start of Turbo Pump [mbar]'
  429 = 'Prevacuum pressure threshold [mbar]'
  92 = 'Prevacuum pressure [mbar]'
  1433 = 'Prevacuum Pressure [mbar]:'
  277 = 'Pulse Tube Year: '
  566 = 'Pump has been running for more than 10 min'
  385 = 'Pump Hours :'
  913 = 'Pump Speed'
  1038 = 'pump speed > 0 rpm'
  740 = 'pump speed > 100 rpm'
  1651 = 'Pump Speed [rpm] :'
  148 = 'Pump State'
  1668 = 'Pump Temp [°C] :'
  1345 = 'PVV1'
  1079 = 'PVV2'
  1190 = 'PVV3'
  115 = 'PVV4'
  34 = 'RAMP'
  302 = 'RE-PRESSURE'
  62 = 'RE-PRESSURISE'
  231 = 'Re-Pressurization'
  379 = 'RE-PRESSURIZE'
  384 = 'Ready :'
  538 = 'Reject [C] :'
  228 = 'Repressure valve'
  75 = 'Root Pump'
  236 = 'Root_OK'
  180 = 'Roughing Pump'
  52 = 'Roughing Pump Speed [rpm]'
  860 = 'rpm'
  12 = 'Running :'
  648 = 'S/N Compressor: '
  952 = 'S/N Panel:'
  754 = 'S/N Pulse Tube: '
  567 = 'Sensor :'
  614 = 'Sensor Name'
  113 = 'Sensor Status'
  542 = 'Set External System command to CLOSE'
  438 = 'Set External System command to OPEN'
  974 = 'Set Points'
  63 = 'SETP'
  442 = 'SetPoint'
  1885 = 'SIM'
  160 = 'Simulated value [K] when simulation is active.'
  2634 = 'Simulated value [mbar] when simulation is active.'
  709 = 'Simulation flag coming from the Control System'
  2496 = 'Simulation flagcoming from the Control System'
  571 = 'Speed > 100 :'
  1446 = 'Standby Speed [rpm] :'
  19 = 'START'
  181 = 'State: '
  401 = 'Status'
  119 = 'STOP'
  156 = 'STOP LN2'
  610 = 'Switch to AUTO Mode'
  1785 = 'Switch to MANUAL Mode'
  590 = 'System Commands'
  924 = 'Target SetPoint'
  623 = 'Target [K] :'
  261 = 'Temperature'
  881 = 'Temperature difference between DET and the coldest point in the Cryostat'
  669 = 'Temperature [°C] :'
  1721 = 'Toggle Engineering Mode'
  1620 = 'Toggle etween Engineering and Commissioning Mode'
  1272 = 'Toggle External System INTERLOCK'
  1622 = 'Turbo Molecular Pump'
  489 = 'Turbo Pump'
  889 = 'Turbo Pump Ready'
  1211 = 'Turbo Pump Speed [rpm]'
  237 = 'Turbo_OK'
  262 = 'Type :'
  645 = 'Underrange'
  404 = 'VAC'
  232 = 'Vac Good'
  478 = 'Vacuum Good'
  400 = 'VAG1'
  647 = 'VAG2'
  1269 = 'VAG3'
  455 = 'VAGF'
  822 = 'VAGF1'
  1083 = 'VAGF2'
  1120 = 'VAGG'
  620 = 'VAGG1'
  812 = 'VAGG2'
  1962 = 'Valid'
  1854 = 'Value used by the system [C]'
  1212 = 'Value used by the system [K]'
  1639 = 'Value used by the system [mbar]'
  681 = 'Valve'
  188 = 'Valve Cmd'
  973 = 'Valve State'
  1494 = 'Valve state: ON=OPEN, OFF=CLOSED'
  621 = 'Valves'
  405 = 'VDC'
  203 = 'WARM-UP'
  35 = 'Warmest Point'
  289 = 'Warmest point in the Cryostat'
  1561 = 'Warning'
  699 = 'Warning :'
  265 = 'Warning if reading is not valid'
  779 = 'Warning if reading is underange. PT100 cannot read below 73.15K (-200C).'
  820 = 'Warning if reading is underrange. PT100 cannot read below 73.15K (-200C).'
  918 = 'Water IN\n%4.1f ºC'
  57 = 'Water OUT\n%4.1f ºC'
  967 = '[%s]'
  912 = '°C'
  1858 = "°C''"
  2136 = '°K'
END_TEXTLIST

// ---- VISUs/GUIs/GUI_ATH2303M_EVAC_LAB.TcVIS
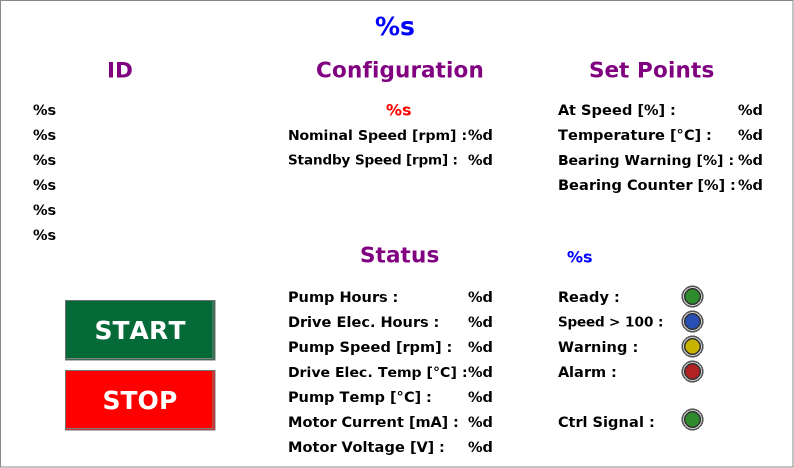
VISUALIZATION GUI_ATH2303M_EVAC_LAB  // 794x468
    Frame (0,0 794x468)
        shows GUI_TEMPLATE_ATH2303M(m_Instance := MAIN.evac_lab.tp, m_bEnable := MAIN.evac_lab.ctrl.bEnable_TP)
END_VISUALIZATION

// ---- VISUs/GUIs/GUI_CMD_OVERRIDE.TcVIS
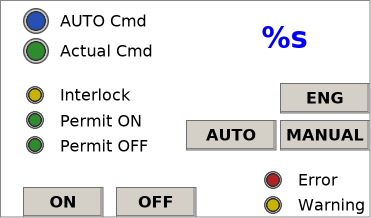
VISUALIZATION GUI_CMD_OVERRIDE  // 371x218
    Frame (0,0 371x218)
        shows GUI_TEMPLATE_CMD_OVERRIDE(m_Cmd := MAIN.cmdOverrideTest)
END_VISUALIZATION

// ---- VISUs/GUIs/GUI_CPA.TcVIS
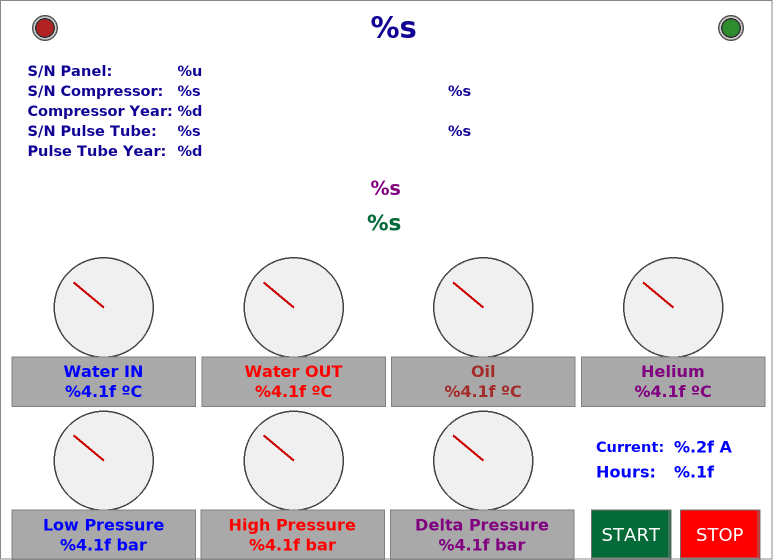
VISUALIZATION GUI_CPA  // 773x560
    Frame (0,0 773x560)
        shows GUI_TEMPLATE_CRYO_CPA(m_Instance := MAIN.Cryo_Ctrl.cpa)
END_VISUALIZATION

// ---- VISUs/GUIs/GUI_CRYO.TcVIS
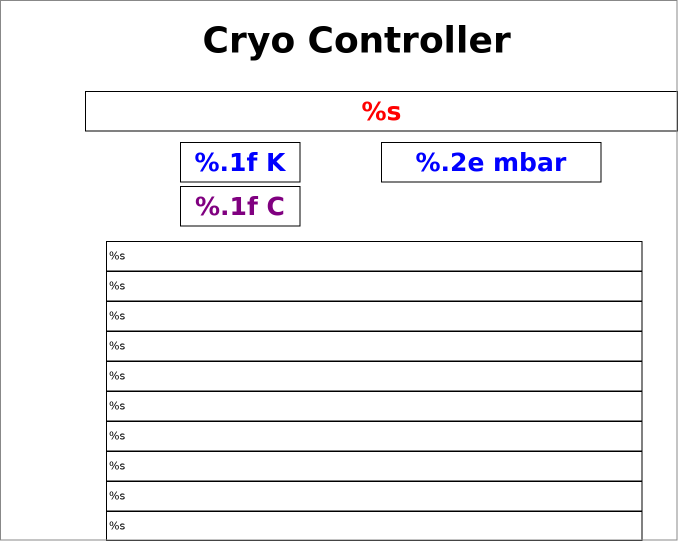
VISUALIZATION GUI_CRYO  // 678x541
    Rectangle (180,142 120x40), "%.1f K", text variable: MAIN.Cryo_Ctrl.Temp_ColdBench.stat.lrTempK
    Rectangle (180,186 120x40), "%.1f C", text variable: MAIN.Cryo_Ctrl.Temp_ColdBench.stat.lrTempC
    Rectangle (381,142 220x40), "%.2e mbar", text variable: MAIN.Cryo_Ctrl.Pressure_Cryo.stat.lrPressure
    Label (182,15 350x50), "Cryo Controller"
    Rectangle (85,91 593x40), "%s", text variable: MAIN.Cryo_Ctrl.stat.sState
    Rectangle (106,241 536x30), "%s", text variable: MAIN.Cryo_Ctrl.syslog.s9
    Rectangle (106,271 536x30), "%s", text variable: MAIN.Cryo_Ctrl.syslog.s8
    Rectangle (106,301 536x30), "%s", text variable: MAIN.Cryo_Ctrl.syslog.s7
    Rectangle (106,331 536x30), "%s", text variable: MAIN.Cryo_Ctrl.syslog.s6
    Rectangle (106,361 536x30), "%s", text variable: MAIN.Cryo_Ctrl.syslog.s5
    Rectangle (106,391 536x30), "%s", text variable: MAIN.Cryo_Ctrl.syslog.s4
    Rectangle (106,421 536x30), "%s", text variable: MAIN.Cryo_Ctrl.syslog.s3
    Rectangle (106,451 536x30), "%s", text variable: MAIN.Cryo_Ctrl.syslog.s2
    Rectangle (106,481 536x30), "%s", text variable: MAIN.Cryo_Ctrl.syslog.s1
    Rectangle (106,511 536x30), "%s", text variable: MAIN.Cryo_Ctrl.syslog.s0
END_VISUALIZATION

// ---- VISUs/GUIs/GUI_CRYOTELGT.TcVIS
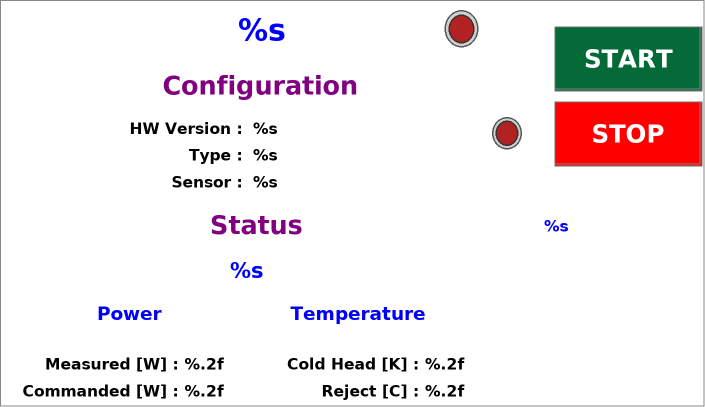
VISUALIZATION GUI_CRYOTELGT  // 705x407
    Frame (0,0 705x407)
        shows GUI_TEMPLATE_CRYOTELGT(m_Instance := MAIN.cooler, m_bEnable := MAIN.bEnable_cooler)
END_VISUALIZATION

// ---- VISUs/GUIs/GUI_ECODRY_V01_EVAC_LAB.TcVIS
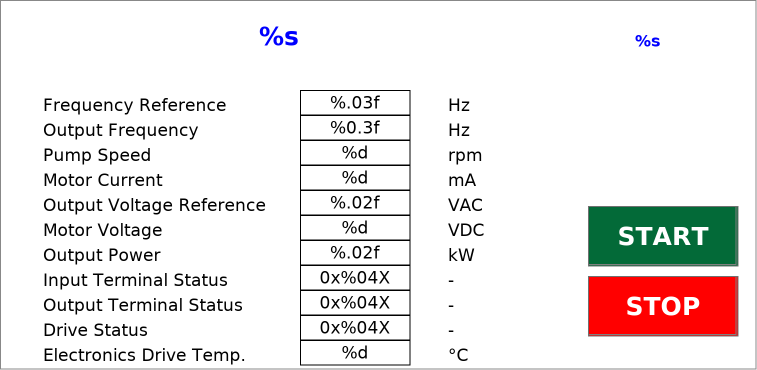
VISUALIZATION GUI_ECODRY_V01_EVAC_LAB  // 757x370
    Frame (0,0 757x370)
        shows GUI_TEMPLATE_ECODRY_V01(m_Instance := MAIN.evac_lab.rp, m_bEnable := MAIN.evac_lab.ctrl.bEnable_RP)
END_VISUALIZATION

// ---- VISUs/GUIs/GUI_EVAC_LAB.TcVIS
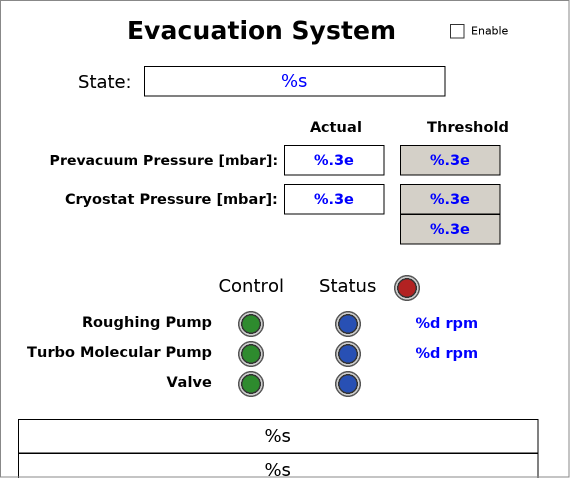
VISUALIZATION GUI_EVAC_LAB  // 570x478
    Frame (0,0 570x478)
        shows GUI_TEMPLATE_CRYO_EVAC_BASE(m_Instance := MAIN.evac_lab, m_bEnable := MAIN.bEnable_evac_lab)
END_VISUALIZATION

// ---- VISUs/GUIs/GUI_EVAC_MICADO.TcVIS
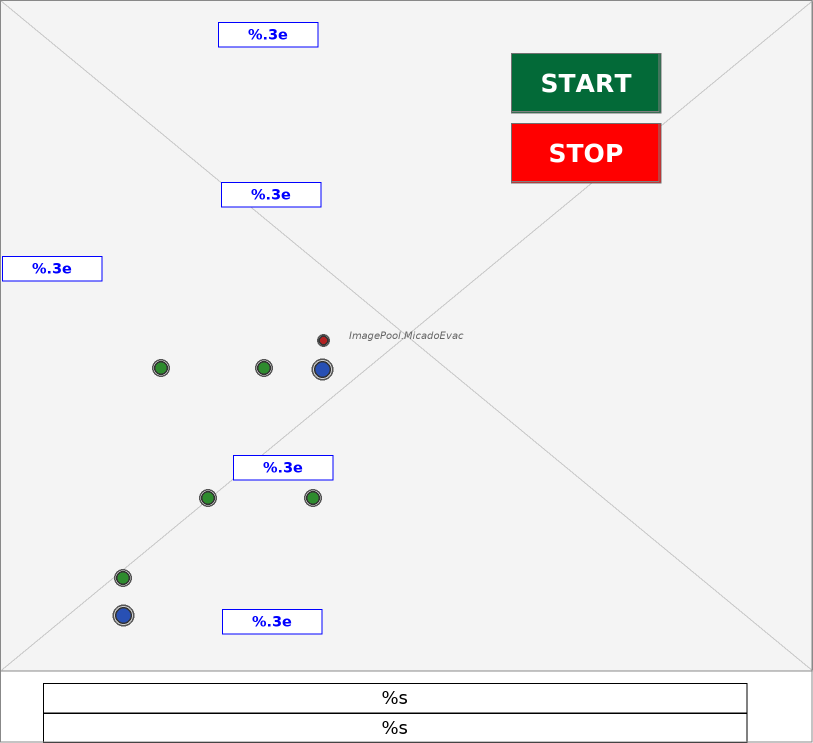
VISUALIZATION GUI_EVAC_MICADO  // 813x743
    Image (0,0 813x671), image: ImagePool.MicadoEvac
    Rectangle (222,609 100x25), "%.3e", text variable: MAIN.evac_micado.VAG1.stat.lrPressure
    Rectangle (233,455 100x25), "%.3e", text variable: MAIN.evac_micado.VAG2.stat.lrPressure
    Rectangle (2,256 100x25), "%.3e", text variable: MAIN.evac_micado.VAG3.stat.lrPressure
    Rectangle (218,22 100x25), "%.3e", text variable: MAIN.evac_micado.VAGF.stat.lrPressure
    Rectangle (221,182 100x25), "%.3e", text variable: MAIN.evac_micado.VAGG.stat.lrPressure
    Lamp1 (111,603 25x25), variable: MAIN.evac_micado.rp.stat.bReady, style: Lamp-Lamp1-Blue
    Lamp1 (310,357 25x25), tooltip "If ON, TMP pump is at its nominal speed, i.e. Ready.", variable: MAIN.evac_micado.tp.stat.bReady, style: Lamp-Lamp1-Blue
    Lamp1 (198,488 20x20), variable: MAIN.evac_micado.PVV1.stat.bActON, style: Lamp-Lamp1-Green
    Lamp1 (303,488 20x20), variable: MAIN.evac_micado.PVV2.stat.bActON, style: Lamp-Lamp1-Green
    Lamp1 (151,358 20x20), variable: MAIN.evac_micado.PVV3.stat.bActON, style: Lamp-Lamp1-Green
    Lamp1 (254,358 20x20), variable: MAIN.evac_micado.PVV4.stat.bActON, style: Lamp-Lamp1-Green
    Lamp1 (113,568 20x20), variable: MAIN.evac_micado.GBV.stat.bActON, style: Lamp-Lamp1-Green
    Rectangle (43,683 704x30), "%s", text variable: MAIN.evac_micado.stat.sErrorText
    Rectangle (43,713 704x30), "%s", text variable: MAIN.evac_micado.stat.sStatus
    Button (511,53 150x60), "START"
        OnMouseClick: execute { MAIN.bEnable_evac_mic := TRUE; }
    Button (511,123 150x60), "STOP"
        OnMouseClick: execute { MAIN.bEnable_evac_mic := FALSE; }
    Lamp1 (316,333 15x15), tooltip "If ON, TMP pump is still spinning.", variable: MAIN.evac_micado.tp.stat.bSpeed100, style: Lamp-Lamp1-Red
END_VISUALIZATION

// ---- VISUs/GUIs/GUI_EVAC_PDS.TcVIS
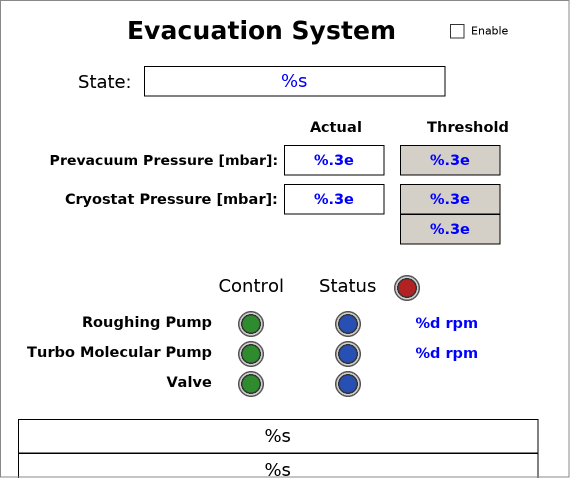
VISUALIZATION GUI_EVAC_PDS  // 570x478
    Frame (0,0 570x478)
        shows GUI_TEMPLATE_CRYO_EVAC_BASE(m_Instance := MAIN.evac_pds, m_bEnable := MAIN.bEnable_evac_pds)
END_VISUALIZATION

// ---- VISUs/GUIs/GUI_HIPACE_30_EVAC_PDS.TcVIS
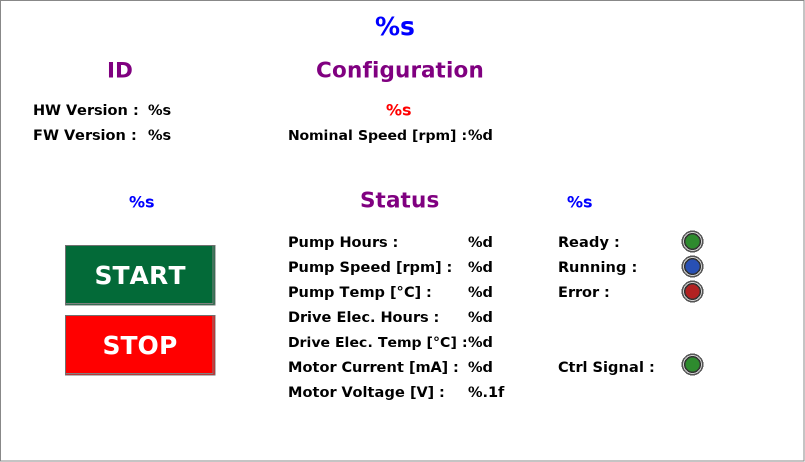
VISUALIZATION GUI_HIPACE_30_EVAC_PDS  // 805x462
    Frame (0,0 805x462)
        shows GUI_TEMPLATE_HIPACE_30(m_Instance := MAIN.evac_pds.tp, m_bEnable := MAIN.evac_pds.ctrl.bEnable_TP)
END_VISUALIZATION

// ---- VISUs/GUIs/GUI_IRATEC.TcVIS
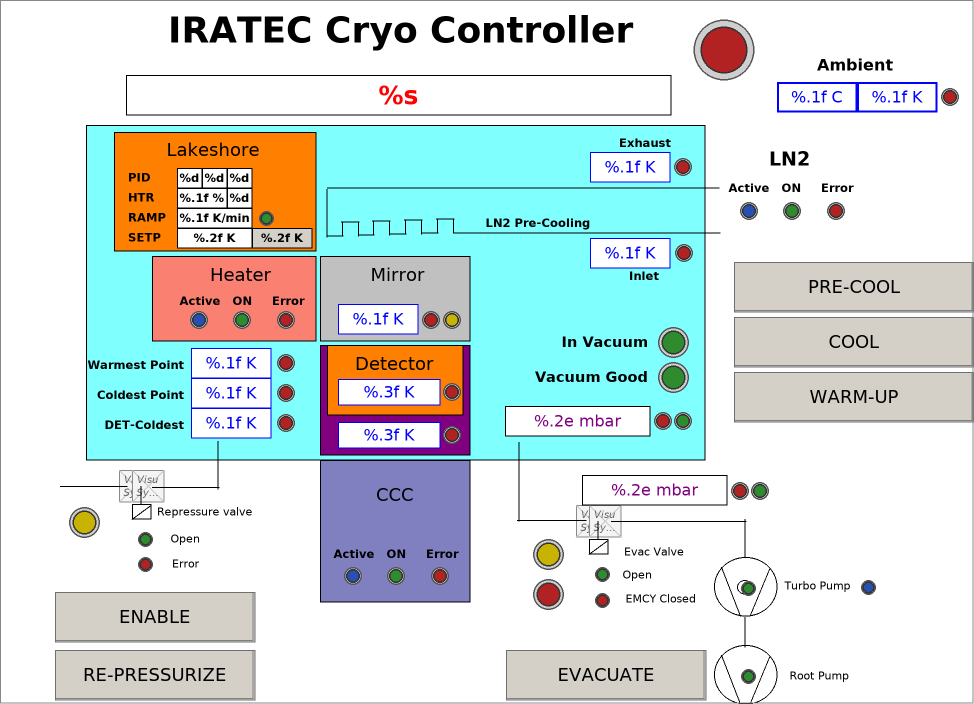
VISUALIZATION GUI_IRATEC  // 974x704
    RoundedRectangle (86,125 619x335)
    Group (327,188 393x50)
        Line (392,0) (0,0)
        Line (0,49) (0,1)
        Line (16,48) (0,48)
        Line (15,34) (15,48)
        Line (32,34) (14,34)
        Line (31,34) (31,48)
        Line (47,47) (31,47)
        Line (46,33) (46,47)
        Line (63,33) (45,33)
        Line (62,33) (62,47)
        Line (79,46) (63,46)
        Line (78,32) (78,46)
        Line (95,32) (77,32)
        Line (94,32) (94,46)
        Line (111,45) (95,45)
        Line (110,31) (110,45)
        Line (127,31) (109,31)
        Line (126,31) (126,45)
        Line (393,45) (126,45)
        Label (136,20 150x30), "LN2 Pre-Cooling"
    Group (714,557 63x59)
        Ellipse (0,0 63x59)
        Ellipse (23,23 15x14)
        Line (7,10) (26,59)
        Line (36,59) (56,11)
    Group (714,645 63x59)
        Ellipse (0,0 63x59)
        Line (7,10) (26,59)
        Line (36,59) (56,11)
    Line (745,647) (745,617)
    Image (576,505 32x32), image: VisuSymbols.Symbols.TriangleRight
    Group (589,505 32x49)
        Image (0,0 32x32), image: VisuSymbols.Symbols.TriangleLeft
        Rectangle (0,34 19x15)
        Line (0,49) (19,35)
        Line (9,34) (9,16)
    Line (745,557) (745,519)
    Line (611,521) (746,521)
    Line (517,520) (586,520)
    Line (519,521) (519,442)
    Rectangle (582,475 145x30), "%.2e mbar", text variable: MAIN.Cryo_Ctrl.Pressure_Evac.stat.lrPressure
    Rectangle (505,406 145x30), "%.2e mbar", text variable: MAIN.Cryo_Ctrl.Pressure_Cryo.stat.lrPressure
    Lamp1 (737,668 23x17), variable: MAIN.Cryo_Ctrl.EvacSys.stat.bRootPumpON, style: Lamp-Lamp1-Green
    Lamp1 (591,566 23x17), variable: MAIN.Cryo_Ctrl.EvacSys.stat.bValveOpen, style: Lamp-Lamp1-Green
    Image (119,470 32x32), image: VisuSymbols.Symbols.TriangleRight
    Group (132,470 32x49)
        Image (0,0 32x32), image: VisuSymbols.Symbols.TriangleLeft
        Rectangle (0,34 19x15)
        Line (0,49) (19,35)
        Line (9,34) (9,16)
    Lamp1 (134,531 23x17), variable: MAIN.Cryo_Ctrl.RepressValve.stat.bActON, style: Lamp-Lamp1-Green
    Line (218,489) (218,441)
    Line (152,487) (219,487)
    Line (60,486) (127,486)
    Label (130,497 150x30), "Repressure valve"
    Label (610,560 55x30), "Open"
    Lamp1 (656,360 35x35), variable: MAIN.Cryo_Ctrl.stat.bGoodVacuum, style: Lamp-Lamp1-Green
    Label (536,362 115x30), "Vacuum Good"
    Label (536,327 115x30), "In Vacuum"
    Lamp1 (656,325 35x35), variable: MAIN.Cryo_Ctrl.stat.bInVacuum, style: Lamp-Lamp1-Green
    Lamp1 (591,592 23x17), variable: MAIN.Cryo_Ctrl.EvacSys.stat.bEmergency, style: Lamp-Lamp1-Red
    Label (609,537 90x30), "Evac Valve"
    Label (614,584 94x30), "EMCY Closed"
    Lamp1 (737,580 23x17), variable: MAIN.Cryo_Ctrl.EvacSys.stat.bTurboPumpON, style: Lamp-Lamp1-Green
    Label (779,661 81x30), "Root Pump"
    Label (777,571 81x30), "Turbo Pump"
    Lamp1 (857,579 23x17), tooltip "Turbo Pump Ready", variable: MAIN.Cryo_Ctrl.EvacSys.stat.bTurboPump10min, style: Lamp-Lamp1-Blue
    Button (506,650 200x50), "EVACUATE", input disabled if: MAIN.Cryo_Ctrl.ctrl.bEnable_RepressSys=TRUE OR MAIN.Cryo_Ctrl.RepressValve.stat.bActON=TRUE
        toggle MAIN.Cryo_Ctrl.ctrl.bEnable_Evac
    Lamp1 (134,556 23x17), variable: MAIN.Cryo_Ctrl.RepressValve.stat.bError, style: Lamp-Lamp1-Red
    Label (158,524 55x30), "Open"
    Label (158,549 55x30), "Error"
    Button (55,592 200x50), "ENABLE", input disabled if: MAIN.Cryo_Ctrl.ctrl.bSafe_Repress=0
        toggle MAIN.Cryo_Ctrl.ctrl.bEnable_RepressSys
    Lamp1 (689,15 70x70), variable: MAIN.Cryo_Ctrl.stat.bError, invisible if: MAIN.Cryo_Ctrl.stat.bError = 0, style: Lamp-Lamp1-Red
    Rectangle (590,238 80x30), "%.1f K", text variable: MAIN.Cryo_Ctrl.Temp_LN2_Inlet.stat.lrTempK
    Rectangle (590,152 80x30), "%.1f K", text variable: MAIN.Cryo_Ctrl.Temp_LN2_Exhaust.stat.lrTempK
    Lamp1 (531,537 35x35), tooltip "If ON, system is enabled", variable: MAIN.Cryo_Ctrl.EvacSys.stat.bEnabled, style: Lamp-Lamp1-Yellow
    Lamp1 (67,505 35x35), tooltip "If ON, system is enabled", variable: MAIN.Cryo_Ctrl.ctrl.bEnable_RepressSys, style: Lamp-Lamp1-Yellow
    Group (716,144 150x77)
        Label (0,29 150x30), "Active ON Error"
        Lamp1 (23,57 20x20), variable: MAIN.Cryo_Ctrl.LN2.stat.bActive, style: Lamp-Lamp1-Blue
        Lamp1 (66,57 20x20), variable: MAIN.Cryo_Ctrl.LN2.stat.bActON, style: Lamp-Lamp1-Green
        Lamp1 (110,57 20x20), variable: MAIN.Cryo_Ctrl.LN2.stat.bError, style: Lamp-Lamp1-Red
        Label (36,0 75x30), "LN2"
    Lamp1 (531,577 35x35), tooltip "If ON, Evacuation System is in ERROR state.", variable: MAIN.Cryo_Ctrl.EvacSys.stat.bError, style: Lamp-Lamp1-Red
    Lamp1 (730,481 20x20), tooltip "Warning if reading is not valid", variable: NOT MAIN.Cryo_Ctrl.EvacSys.in_Pressure_Evac.bValid, style: Lamp-Lamp1-Red
    Group (320,460 151x142)
        Rectangle (0,0 150x142), "CCC"
        Lamp1 (23,106 20x20), tooltip "CCC Control is Enabled/Active", variable: MAIN.Cryo_Ctrl.CCC.stat.bActive, style: Lamp-Lamp1-Blue
        Lamp1 (66,106 20x20), tooltip "CCC is ON", variable: MAIN.Cryo_Ctrl.CCC.stat.bActON, style: Lamp-Lamp1-Green
        Lamp1 (110,106 20x20), variable: MAIN.Cryo_Ctrl.CCC.stat.bError, style: Lamp-Lamp1-Red
        Label (1,79 150x30), "Active ON Error"
    Label (602,128 86x30), "Exhaust"
    Label (601,261 86x30), "Inlet"
    Lamp1 (673,157 20x20), tooltip "Warning if reading is not valid", variable: NOT MAIN.Cryo_Ctrl.Temp_LN2_Exhaust.stat.bValid, style: Lamp-Lamp1-Red
    Lamp1 (674,243 20x20), tooltip "Warning if reading is not valid", variable: NOT MAIN.Cryo_Ctrl.Temp_LN2_Inlet.stat.bValid, style: Lamp-Lamp1-Red
    Lamp1 (653,411 20x20), tooltip "Warning if reading is not valid", variable: NOT MAIN.Cryo_Ctrl.Pressure_Cryo.stat.bValid, style: Lamp-Lamp1-Red
    Button (55,650 200x50), "RE-PRESSURIZE", input disabled if: MAIN.Cryo_Ctrl.ctrl.bEnable_RepressSys=0
        toggle MAIN.Cryo_Ctrl.ctrl.bEnable_RepressCtrl
    Button (734,262 240x50), "PRE-COOL", input disabled if: MAIN.Cryo_Ctrl.ctrl.bSafe_Precool = 0
        toggle MAIN.Cryo_Ctrl.ctrl.bEnable_Precool
    Button (734,317 240x50), "COOL", input disabled if: MAIN.Cryo_Ctrl.ctrl.bSafe_Cooling=0
        toggle MAIN.Cryo_Ctrl.ctrl.bEnable_Cool
    Button (734,372 240x50), "WARM-UP", input disabled if: MAIN.Cryo_Ctrl.ctrl.bSafe_Warmup=0
        toggle MAIN.Cryo_Ctrl.ctrl.bEnable_Warmup
    Label (152,5 498x50), "IRATEC Cryo Controller"
    Rectangle (126,75 545x40), "%s", text variable: MAIN.Cryo_Ctrl.stat.sState
    Group (152,256 165x85)
        Rectangle (0,0 164x85)
        Label (15,30 150x30), "Active ON Error"
        Lamp1 (37,54 20x20), tooltip "Heater Control is Enabled/Active", variable: MAIN.Cryo_Ctrl.Heater.stat.bActive, style: Lamp-Lamp1-Blue
        Lamp1 (80,54 20x20), tooltip "Heater is ON", variable: MAIN.Cryo_Ctrl.Heater.stat.bActON, style: Lamp-Lamp1-Green
        Lamp1 (124,54 20x20), variable: MAIN.Cryo_Ctrl.Heater.stat.bError, style: Lamp-Lamp1-Red
        Label (47,4 83x30), "Heater"
    Lamp1 (750,481 20x20), tooltip "Flag if reading is in sensor range", variable: MAIN.Cryo_Ctrl.EvacSys.in_Pressure_Evac.bInRange, style: Lamp-Lamp1-Green
    Lamp1 (673,411 20x20), tooltip "Flag if reading is in sensor range", variable: MAIN.Cryo_Ctrl.EvacSys.in_Pressure_Cryo.bInRange, style: Lamp-Lamp1-Green
    Label (92,380 95x30), "Coldest Point"
    Rectangle (191,378 80x30), "%.1f K", tooltip "Coldest point in the Cryostat", text variable: MAIN.Cryo_Ctrl.stat.lrLowestTempK
    Lamp1 (276,383 20x20), tooltip "Warning if reading is not valid", variable: NOT MAIN.Cryo_Ctrl.stat.bLowestTempValid, style: Lamp-Lamp1-Red
    Rectangle (191,408 80x30), "%.1f K", tooltip "Temperature difference between DET and the coldest point in the Cryostat", text variable: MAIN.Cryo_Ctrl.stat.lrDiffTempK
    Label (92,410 95x30), "DET-Coldest"
    Lamp1 (276,413 20x20), tooltip "Warning if reading is not valid", variable: NOT MAIN.Cryo_Ctrl.stat.bDiffTempValid, style: Lamp-Lamp1-Red
    Label (92,350 95x30), "Warmest Point"
    Rectangle (191,348 80x30), "%.1f K", tooltip "Warmest point in the Cryostat", text variable: MAIN.Cryo_Ctrl.stat.lrHighestTempK
    Lamp1 (276,353 20x20), tooltip "Warning if reading is not valid", variable: NOT MAIN.Cryo_Ctrl.stat.bHighestTempValid, style: Lamp-Lamp1-Red
    Rectangle (114,132 202x119)
    Label (160,135 106x30), "Lakeshore"
    Label (125,170 40x15), "PID"
    Label (125,190 40x15), "HTR"
    Label (125,210 40x15), "RAMP"
    Label (125,230 40x15), "SETP"
    Rectangle (177,168 25x20), "%d", text variable: MAIN.Cryo_Ctrl.Lakeshore.stat.nPID_P
    Rectangle (202,168 25x20), "%d", text variable: MAIN.Cryo_Ctrl.Lakeshore.stat.nPID_I
    Rectangle (227,168 25x20), "%d", text variable: MAIN.Cryo_Ctrl.Lakeshore.stat.nPID_D
    Rectangle (177,188 50x20), "%.1f %", tooltip "Heater Output [%]", text variable: MAIN.Cryo_Ctrl.Lakeshore.stat.lrHTR
    Rectangle (177,208 75x20), "%.1f K/min", tooltip "Heater Ramp Rate", text variable: MAIN.Cryo_Ctrl.Lakeshore.stat.lrRAMP_Rate
    Lamp1 (255,210 23x17), tooltip "Flag if Heater RAMP is On", variable: MAIN.Cryo_Ctrl.Lakeshore.stat.bRAMP_On, style: Lamp-Lamp1-Green
    Rectangle (177,228 75x20), "%.2f K", tooltip "SetPoint", text variable: MAIN.Cryo_Ctrl.Lakeshore.stat.lrSETP
    Rectangle (227,188 25x20), "%d", tooltip "Heater Range", text variable: MAIN.Cryo_Ctrl.Lakeshore.stat.nRANGE
    Group (320,256 150x85)
        Rectangle (0,0 150x85)
        Label (29,4 97x30), "Mirror"
        Rectangle (18,48 80x30), "%.1f K", text variable: MAIN.Cryo_Ctrl.Temp_Mirror.stat.lrTempK
        Lamp1 (101,54 20x20), tooltip "Warning if reading is not valid", variable: NOT MAIN.Cryo_Ctrl.Temp_Mirror.stat.bValid, style: Lamp-Lamp1-Red
        Lamp1 (122,54 20x20), tooltip "Warning if reading is underrange. PT100 cannot read below 73.15K (-200C).", variable: NOT MAIN.Cryo_Ctrl.Temp_Mirror.stat.bInRange, style: Lamp-Lamp1-Yellow
    Group (320,345 150x110)
        Rectangle (0,0 150x110)
        Rectangle (18,77 102x26), "%.3f K", tooltip "Heat Shield Temperature", text variable: MAIN.Cryo_Ctrl.Temp_HeatShield.stat.lrTempK
        Lamp1 (122,80 20x20), tooltip "Warning if reading is not valid", variable: NOT MAIN.Cryo_Ctrl.Temp_HeatShield.stat.bValid, style: Lamp-Lamp1-Red
    Group (327,345 136x70)
        Rectangle (0,0 136x70)
        Rectangle (11,34 102x26), "%.3f K", text variable: MAIN.Cryo_Ctrl.Temp_DET.stat.lrTempK
        Lamp1 (115,37 20x20), tooltip "Warning if reading is not valid", variable: NOT MAIN.Cryo_Ctrl.Temp_DET.stat.bValid, style: Lamp-Lamp1-Red
        Label (26,4 83x30), "Detector"
    Rectangle (252,228 60x20), "%.2f K", tooltip "Target SetPoint", text variable: MAIN.Cryo_Ctrl.Lakeshore.stat.lrSETP_Target
    Rectangle (857,82 80x30), "%.1f K", text variable: MAIN.Cryo_Ctrl.Temp_Ambient.stat.lrTempK
    Lamp1 (940,87 20x20), tooltip "Warning if reading is not valid", variable: NOT MAIN.Cryo_Ctrl.Temp_Ambient.stat.bValid, style: Lamp-Lamp1-Red
    Rectangle (777,82 80x30), "%.1f C", text variable: MAIN.Cryo_Ctrl.Temp_Ambient.stat.lrTempC
    Label (812,50 86x30), "Ambient"
END_VISUALIZATION

// ---- VISUs/GUIs/GUI_MICADO_Valves.TcVIS
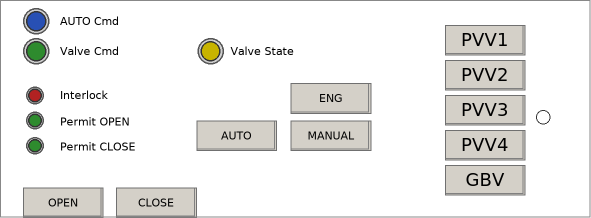
VISUALIZATION GUI_MICADO_Valves  // 591x218
    Frame (0,0 371x218)
        shows GUI_TEMPLATE_ACTUATOR_ENG(m_Cmd := MAIN.evac_micado.ptrVC[MAIN.evac_micado.guiValveIndex]^, m_Valve := MAIN.evac_micado.ptrV[MAIN.evac_micado.guiValveIndex]^)
    Button (445,25 80x30), "PVV1"
        OnMouseClick: execute { MAIN.evac_micado.guiValveIndex := 1; }
    Button (445,60 80x30), "PVV2"
        OnMouseClick: execute { MAIN.evac_micado.guiValveIndex := 2; }
    Button (445,95 80x30), "PVV3"
        OnMouseClick: execute { MAIN.evac_micado.guiValveIndex := 3; }
    Button (445,130 80x30), "PVV4"
        OnMouseClick: execute { MAIN.evac_micado.guiValveIndex := 4; }
    Button (445,165 80x30), "GBV"
        OnMouseClick: execute { MAIN.evac_micado.guiValveIndex := 5; }
    RadioButton (534,28 57x178), variable: MAIN.evac_micado.guiValveIndex-1
END_VISUALIZATION

// ---- VISUs/GUIs/GUI_MVP030_EVAC_PDS.TcVIS
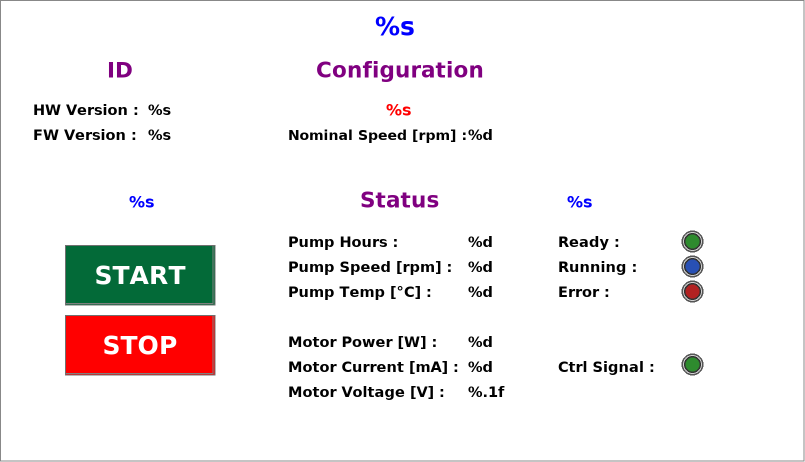
VISUALIZATION GUI_MVP030_EVAC_PDS  // 805x462
    Frame (0,0 805x462)
        shows GUI_TEMPLATE_MVP030(m_Instance := MAIN.evac_pds.rp, m_bEnable := MAIN.evac_pds.ctrl.bEnable_RP)
END_VISUALIZATION

// ---- VISUs/GUIs/GUI_P2_OVERRIDE.TcVIS
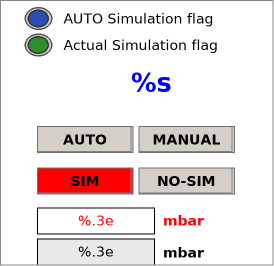
VISUALIZATION GUI_P2_OVERRIDE  // 274x266
    Frame (0,0 274x266)
        shows GUI_TEMPLATE_PRESS_OVERRIDE(m_Cmd := MAIN.pressOR_P1, m_Press := MAIN.P1)
END_VISUALIZATION

// ---- VISUs/GUIs/GUI_Pressures.TcVIS
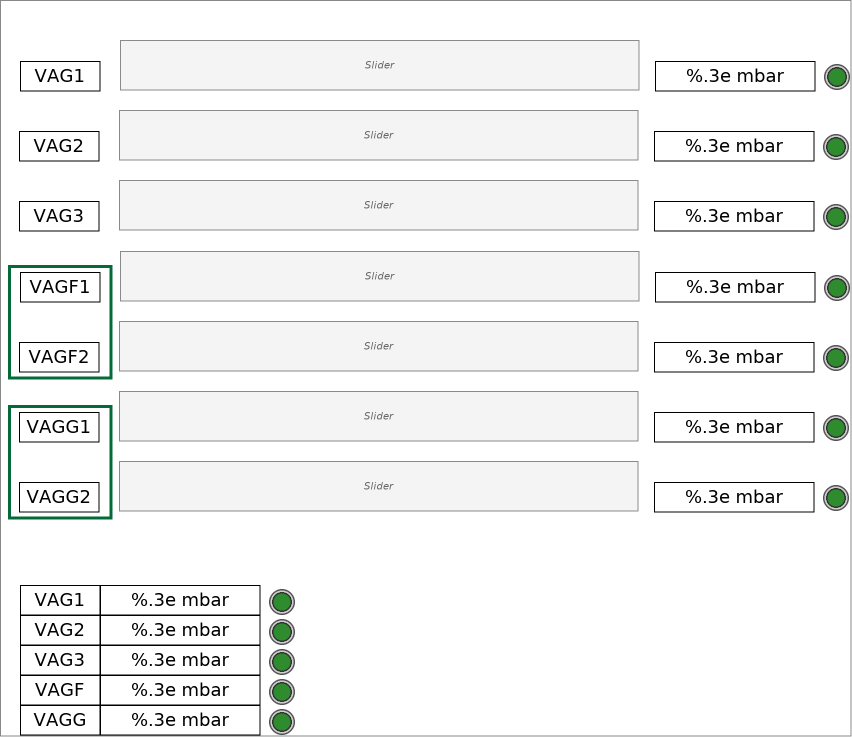
VISUALIZATION GUI_Pressures  // 852x737
    Slider (120,40 519x50), variable: MAIN.q_nVAG1, scale 0..35000
    Rectangle (20,61 80x30), "VAG1"
    Rectangle (655,61 160x30), "%.3e mbar", text variable: MAIN.evac_micado.VAG1.stat.lrPressure
    Lamp1 (822,62 30x30), variable: MAIN.evac_micado.VAG1.stat.bValid, style: Lamp-Lamp1-Green
    Slider (119,110 519x50), variable: MAIN.q_nVAG2, scale 0..35000
    Rectangle (19,131 80x30), "VAG2"
    Rectangle (654,131 160x30), "%.3e mbar", text variable: MAIN.evac_micado.VAG2.stat.lrPressure
    Lamp1 (821,132 30x30), variable: MAIN.evac_micado.VAG2.stat.bValid, style: Lamp-Lamp1-Green
    Slider (119,180 519x50), variable: MAIN.q_nVAG3, scale 0..35000
    Rectangle (19,201 80x30), "VAG3"
    Rectangle (654,201 160x30), "%.3e mbar", text variable: MAIN.evac_micado.VAG3.stat.lrPressure
    Lamp1 (821,202 30x30), variable: MAIN.evac_micado.VAG3.stat.bValid, style: Lamp-Lamp1-Green
    Slider (120,251 519x50), variable: MAIN.q_nVAGF1, scale 0..35000
    Rectangle (20,272 80x30), "VAGF1"
    Rectangle (655,272 160x30), "%.3e mbar", text variable: MAIN.sensor_VAGF1.stat.lrPressure
    Lamp1 (822,273 30x30), variable: MAIN.sensor_VAGF1.stat.bValid, style: Lamp-Lamp1-Green
    Slider (119,321 519x50), variable: MAIN.q_nVAGF2, scale 0..35000
    Rectangle (19,342 80x30), "VAGF2"
    Rectangle (654,342 160x30), "%.3e mbar", text variable: MAIN.sensor_VAGF2.stat.lrPressure
    Lamp1 (821,343 30x30), variable: MAIN.sensor_VAGF2.stat.bValid, style: Lamp-Lamp1-Green
    Slider (119,391 519x50), variable: MAIN.q_nVAGG1, scale 0..35000
    Rectangle (19,412 80x30), "VAGG1"
    Rectangle (654,412 160x30), "%.3e mbar", text variable: MAIN.sensor_VAGG1.stat.lrPressure
    Lamp1 (821,413 30x30), variable: MAIN.sensor_VAGG1.stat.bValid, style: Lamp-Lamp1-Green
    Slider (119,461 519x50), variable: MAIN.q_nVAGG2, scale 0..35000
    Rectangle (19,482 80x30), "VAGG2"
    Rectangle (654,482 160x30), "%.3e mbar", text variable: MAIN.sensor_VAGG2.stat.lrPressure
    Lamp1 (821,483 30x30), variable: MAIN.sensor_VAGG2.stat.bValid, style: Lamp-Lamp1-Green
    Rectangle (20,585 80x30), "VAG1"
    Rectangle (20,615 80x30), "VAG2"
    Rectangle (20,645 80x30), "VAG3"
    Rectangle (100,585 160x30), "%.3e mbar", text variable: MAIN.evac_micado.VAG1.stat.lrPressure
    Lamp1 (267,587 30x30), variable: MAIN.evac_micado.VAG1.stat.bValid, style: Lamp-Lamp1-Green
    Rectangle (100,615 160x30), "%.3e mbar", text variable: MAIN.evac_micado.VAG2.stat.lrPressure
    Lamp1 (267,617 30x30), variable: MAIN.evac_micado.VAG2.stat.bValid, style: Lamp-Lamp1-Green
    Rectangle (100,645 160x30), "%.3e mbar", text variable: MAIN.evac_micado.VAG3.stat.lrPressure
    Lamp1 (267,647 30x30), variable: MAIN.evac_micado.VAG3.stat.bValid, style: Lamp-Lamp1-Green
    Rectangle (20,675 80x30), "VAGF"
    Rectangle (100,675 160x30), "%.3e mbar", text variable: MAIN.evac_micado.VAGF.stat.lrPressure
    Lamp1 (267,677 30x30), variable: MAIN.evac_micado.VAGF.stat.bValid, style: Lamp-Lamp1-Green
    Rectangle (20,705 80x30), "VAGG"
    Rectangle (100,705 160x30), "%.3e mbar", text variable: MAIN.evac_micado.VAGG.stat.lrPressure
    Lamp1 (267,707 30x30), variable: MAIN.evac_micado.VAGG.stat.bValid, style: Lamp-Lamp1-Green
    Rectangle (8,265 104x114)
    Rectangle (8,405 104x114)
END_VISUALIZATION

// ---- VISUs/GUIs/GUI_PVV1_CMD.TcVIS
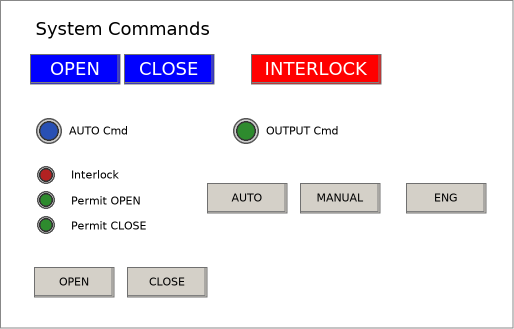
VISUALIZATION GUI_PVV1_CMD  // 514x329
    Frame (11,105 503x224)
        shows GUI_TEMPLATE_ACTUATOR_CMD(m_Instance := MAIN.cmdPVV1)
    Button (30,54 90x30), "OPEN", tooltip "Set External System command to OPEN"
        OnMouseClick: execute { MAIN.bCmdPVV1 := TRUE; }
    Button (124,54 90x30), "CLOSE", tooltip "Set External System command to CLOSE"
        OnMouseClick: execute { MAIN.bCmdPVV1 := FALSE; }
    Rectangle (33,14 180x30), "System Commands"
    Button (251,54 130x30), "INTERLOCK", tooltip "Toggle External System INTERLOCK"
        toggle MAIN.bIntlkPVV1
        OnMouseClick: execute { MAIN.bCmdPVV1 := TRUE; }
END_VISUALIZATION

// ---- VISUs/GUIs/GUI_SBG232.TcVIS
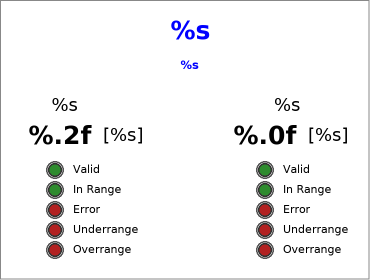
VISUALIZATION GUI_SBG232  // 370x280
    Frame (0,0 370x280)
        shows GUI_TEMPLATE_SBG232(m_Instance := MAIN.sbg232)
END_VISUALIZATION

// ---- VISUs/GUIs/GUI_SBG232_SIM.TcVIS
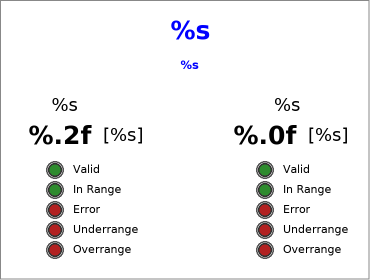
VISUALIZATION GUI_SBG232_SIM  // 370x280
    Frame (0,0 370x280)
        shows GUI_TEMPLATE_SBG232(m_Instance := MAIN.sbg232_sim)
END_VISUALIZATION

// ---- VISUs/GUIs/GUI_T2_OVERRIDE.TcVIS
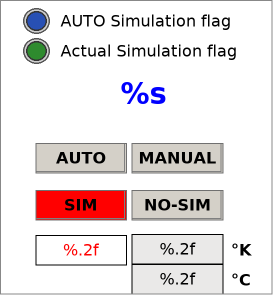
VISUALIZATION GUI_T2_OVERRIDE  // 273x295
    Frame (0,0 273x295)
        shows GUI_TEMPLATE_TEMP_OVERRIDE(m_Cmd := MAIN.tempOR_T2, m_Temp := MAIN.T2)
END_VISUALIZATION

// ---- VISUs/Templates/GUI_TEMPLATE_ACTUATOR_CMD.TcVIS
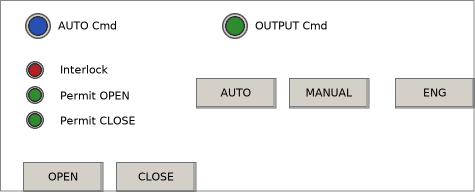
VISUALIZATION GUI_TEMPLATE_ACTUATOR_CMD  // 475x192
VAR_IN_OUT
	m_Instance:	FB_CRYO_ACTUATOR_CMD;
END_VAR
    Lamp1 (25,60 20x20), variable: m_Instance.in_bInterlock, style: Lamp-Lamp1-Red
    Lamp1 (25,85 20x20), variable: m_Instance.bPermitOn, style: Lamp-Lamp1-Green
    Lamp1 (25,110 20x20), variable: m_Instance.bPermitOff, style: Lamp-Lamp1-Green
    Rectangle (57,55 83x30), "Interlock"
    Rectangle (57,81 83x30), "Permit OPEN"
    Rectangle (57,106 83x30), "Permit CLOSE"
    Button (23,162 80x30), "OPEN", colour toggle: (m_Instance.bPermitOn AND NOT m_Instance.bAutoMode) OR m_Instance.bEngMode, input disabled if: m_Instance.bDisableBtnOn
        OnMouseClick: execute { m_Instance.bManualCmd := TRUE; m_Instance.bManualExecute := TRUE; }
    Lamp1 (220,11 30x30), variable: m_Instance.out_Enable, style: Lamp-Lamp1-Green
    Rectangle (252,11 83x30), "OUTPUT Cmd"
    Button (196,78 80x30), "AUTO", colour toggle: m_Instance.bAutoMode, input disabled if: m_Instance.bAutoMode OR m_Instance.bEngMode
        OnMouseClick: execute { m_Instance.bAutoMode := TRUE; }
    Button (289,78 80x30), "MANUAL", colour toggle: NOT m_Instance.bAutoMode, input disabled if: NOT m_Instance.bAutoMode AND NOT_IDLE m_Instance.bEngMode
        OnMouseClick: execute { m_Instance.bAutoMode := FALSE; }
    Button (116,162 80x30), "CLOSE", colour toggle: (m_Instance.bPermitOff AND NOT m_Instance.bAutoMode) OR m_Instance.bEngMode, input disabled if: m_Instance.bDisableBtnOff
        OnMouseClick: execute { m_Instance.bManualCmd := FALSE; m_Instance.bManualExecute := TRUE; }
    Button (395,78 80x30), "ENG", tooltip "Engineering / Commissioning Mode", colour toggle: m_Instance.bEngMode, input disabled if: m_Instance.bAutoMode
        toggle m_Instance.bEngMode
    Lamp1 (23,11 30x30), variable: m_Instance.in_bEnable, style: Lamp-Lamp1-Blue
    Rectangle (55,11 83x30), "AUTO Cmd"
END_VISUALIZATION

// ---- VISUs/Templates/GUI_TEMPLATE_ACTUATOR_ENG.TcVIS
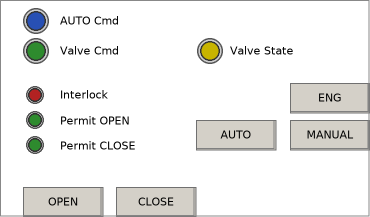
VISUALIZATION GUI_TEMPLATE_ACTUATOR_ENG  // 370x217
VAR_IN_OUT
	m_Cmd:		FB_CRYO_ACTUATOR_CMD;
	m_Valve:	FB_CRYO_VALVE_CTRL;
END_VAR
    Lamp1 (25,85 20x20), variable: m_Cmd.in_bInterlock, style: Lamp-Lamp1-Red
    Lamp1 (25,110 20x20), variable: m_Cmd.bPermitOn, style: Lamp-Lamp1-Green
    Lamp1 (25,135 20x20), variable: m_Cmd.bPermitOff, style: Lamp-Lamp1-Green
    Rectangle (57,80 83x30), "Interlock"
    Rectangle (57,106 83x30), "Permit OPEN"
    Rectangle (57,131 83x30), "Permit CLOSE"
    Button (23,187 80x30), "OPEN", colour toggle: (m_Cmd.bPermitOn AND NOT m_Cmd.bAutoMode) OR m_Cmd.bEngMode, input disabled if: m_Cmd.bDisableBtnOn
        OnMouseClick: execute { m_Cmd.bManualCmd := TRUE; m_Cmd.bManualExecute := TRUE; }
    Lamp1 (21,36 30x30), tooltip "Actual Valve command", variable: m_Cmd.out_bEnable, style: Lamp-Lamp1-Green
    Rectangle (57,36 83x30), "Valve Cmd"
    Button (196,120 80x30), "AUTO", colour toggle: m_Cmd.bAutoMode, input disabled if: m_Cmd.bAutoMode OR m_Cmd.bEngMode
        OnMouseClick: execute { m_Cmd.bAutoMode := TRUE; }
    Button (290,120 80x30), "MANUAL", colour toggle: NOT m_Cmd.bAutoMode, input disabled if: NOT m_Cmd.bAutoMode AND NOT m_Cmd.bEngMode
        OnMouseClick: execute { m_Cmd.bAutoMode := FALSE; }
    Button (116,187 80x30), "CLOSE", colour toggle: (m_Cmd.bPermitOff AND NOT m_Cmd.bAutoMode) OR m_Cmd.bEngMode, input disabled if: m_Cmd.bDisableBtnOff
        OnMouseClick: execute { m_Cmd.bManualCmd := FALSE; m_Cmd.bManualExecute := TRUE; }
    Button (290,83 80x30), "ENG", tooltip "Engineering / Commissioning Mode", colour toggle: m_Cmd.bEngMode, input disabled if: m_Cmd.bAutoMode
        toggle m_Cmd.bEngMode
    Lamp1 (21,6 30x30), tooltip "Command coming from the Control System", variable: m_Cmd.in_bEnable, style: Lamp-Lamp1-Blue
    Rectangle (57,6 83x30), "AUTO Cmd"
    Lamp1 (195,36 30x30), tooltip "Valve state: ON=OPEN, OFF=CLOSED", variable: m_Valve.stat.bActON, style: Lamp-Lamp1-Yellow
    Rectangle (227,36 83x30), "Valve State"
END_VISUALIZATION

// ---- VISUs/Templates/GUI_TEMPLATE_SENSOR_SIM_OVERRIDE.TcVIS
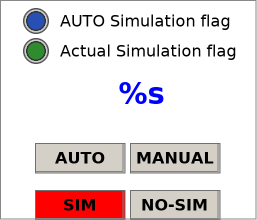
VISUALIZATION GUI_TEMPLATE_SENSOR_SIM_OVERRIDE  // 257x220
VAR_IN_OUT
	m_Cmd:		FB_CRYO_CMD_OVERRIDE;
END_VAR
    Button (35,190 90x30), "SIM", tooltip "Activate Simulation", colour toggle: (m_Cmd.bPermitOn AND NOT m_Cmd.bAutoMode) OR m_Cmd.bEngMode, input disabled if: m_Cmd.bDisableBtnOn
        OnMouseClick: execute { m_Cmd.bManualCmd := TRUE; }
    Lamp1 (21,36 30x30), tooltip "Actual command going out", variable: m_Cmd.out_bEnable, style: Lamp-Lamp1-Green
    Rectangle (57,36 200x30), "Actual Simulation flag", tooltip "Actual Simulation flag set the user"
    Button (35,143 90x30), "AUTO", tooltip "Switch to AUTO Mode", colour toggle: m_Cmd.bAutoMode, input disabled if: m_Cmd.bAutoMode OR m_Cmd.bEngMode
        OnMouseClick: execute { m_Cmd.bAutoMode := TRUE; }
    Button (130,143 90x30), "MANUAL", tooltip "Switch to MANUAL Mode", colour toggle: NOT m_Cmd.bAutoMode, input disabled if: NOT m_Cmd.bAutoMode AND NOT m_Cmd.bEngMode
        OnMouseClick: execute { m_Cmd.bAutoMode := FALSE; }
    Button (130,190 90x30), "NO-SIM", tooltip "Deactivate Simulation", colour toggle: (m_Cmd.bPermitOff AND NOT m_Cmd.bAutoMode) OR m_Cmd.bEngMode, input disabled if: m_Cmd.bDisableBtnOff
        OnMouseClick: execute { m_Cmd.bManualCmd := FALSE; }
    Lamp1 (21,6 30x30), tooltip "Simulation flagcoming from the Control System", variable: m_Cmd.in_bEnable, style: Lamp-Lamp1-Blue
    Rectangle (57,6 200x30), "AUTO Simulation flag", tooltip "AUTO Simulation flag set by the system"
    Rectangle (67,73 150x41), "%s", text variable: m_Cmd.out_sMode
END_VISUALIZATION

// ---- VISUs/Templates/GUI_TEMPLATE_ATH2303M.TcVIS
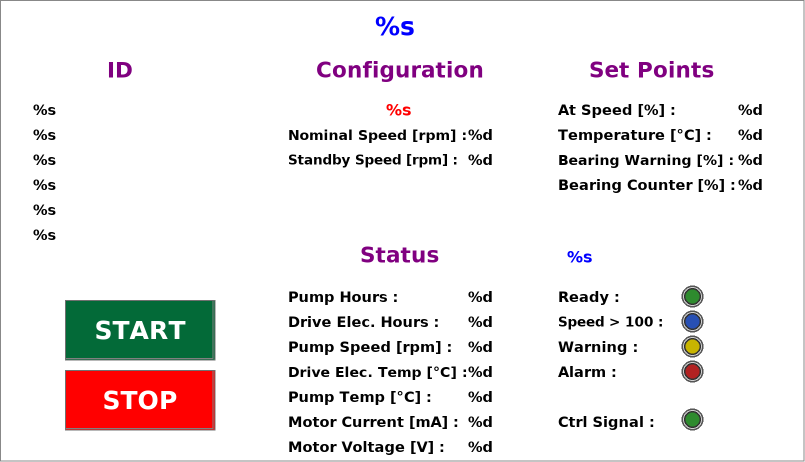
VISUALIZATION GUI_TEMPLATE_ATH2303M  // 805x462
VAR_IN_OUT
	m_Instance:	FB_CRYO_PUMP_ATH2303M;
	m_bEnable:	BOOL;	// Flag to start/stop the pump
END_VAR
    Rectangle (45,55 150x30), "ID"
    Rectangle (310,55 180x30), "Configuration"
    Rectangle (325,240 150x30), "Status"
    Lamp1 (680,284 25x25), tooltip "OK for Process, i.e. speed ≥ nominal speed", variable: m_Instance.stat.bReady, style: Lamp-Lamp1-Green
    Lamp1 (680,309 25x25), tooltip "pump speed > 100 rpm", variable: m_Instance.stat.bSpeed100, style: Lamp-Lamp1-Blue
    Lamp1 (680,334 25x25), tooltip "presence of a warning", variable: m_Instance.stat.bWarning, style: Lamp-Lamp1-Yellow
    Lamp1 (680,359 25x25), tooltip "presence of an alarm", variable: m_Instance.stat.bAlarm, style: Lamp-Lamp1-Red
    Rectangle (555,282 110x30), "Ready :"
    Rectangle (555,307 110x30), "Speed > 100 :"
    Rectangle (555,332 110x30), "Warning :"
    Rectangle (555,357 110x30), "Alarm :"
    Rectangle (30,145 240x30), "%s", text variable: m_Instance.stat.sVer1
    Rectangle (30,170 240x30), "%s", text variable: m_Instance.stat.sVer2
    Rectangle (30,195 240x30), "%s", text variable: m_Instance.stat.sVer3
    Rectangle (30,220 240x30), "%s", text variable: m_Instance.stat.sVer4
    Rectangle (285,120 180x30), "Nominal Speed [rpm] :"
    Rectangle (285,145 180x30), "Standby Speed [rpm] :"
    Rectangle (285,282 180x30), "Pump Hours :"
    Rectangle (285,307 180x30), "Drive Elec. Hours :"
    Rectangle (577,55 150x30), "Set Points"
    Rectangle (555,95 180x30), "At Speed [%] :"
    Rectangle (555,120 180x30), "Temperature [°C] :"
    Rectangle (555,145 180x30), "Bearing Warning [%] :"
    Rectangle (555,170 180x30), "Bearing Counter [%] :"
    Rectangle (735,95 70x30), "%d", text variable: m_Instance.stat.nSetPoint_AtSpeed
    Rectangle (735,120 70x30), "%d", text variable: m_Instance.stat.nSetPoint_Temp
    Rectangle (735,145 70x30), "%d", text variable: m_Instance.stat.nSetPoint_BearingWarn
    Rectangle (735,170 70x30), "%d", text variable: m_Instance.stat.nSetPoint_BearingCounter
    Rectangle (465,120 70x30), "%d", text variable: m_Instance.stat.nNominalSpeed
    Rectangle (465,145 70x30), "%d", text variable: m_Instance.stat.nStandbySpeed
    Rectangle (465,282 70x30), "%d", text variable: m_Instance.stat.nPumpHours
    Rectangle (465,307 70x30), "%d", text variable: m_Instance.stat.nElecHours
    Rectangle (285,332 180x30), "Pump Speed [rpm] :"
    Rectangle (465,332 70x30), "%d", text variable: m_Instance.stat.nPumpSpeed
    Rectangle (285,357 180x30), "Drive Elec. Temp [°C] :"
    Rectangle (465,357 70x30), "%d", text variable: m_Instance.stat.nElecTemp
    Rectangle (285,382 180x30), "Pump Temp [°C] :"
    Rectangle (465,382 70x30), "%d", text variable: m_Instance.stat.nPumpTemp
    Rectangle (285,407 180x30), "Motor Current [mA] :"
    Rectangle (465,407 70x30), "%d", text variable: m_Instance.stat.nMotorCurr
    Rectangle (285,432 180x30), "Motor Voltage [V] :"
    Rectangle (465,432 70x30), "%d", text variable: m_Instance.stat.nMotorVolt
    Rectangle (280,11 230x30), "%s", text variable: m_Instance.in_sName
    Rectangle (289,95 220x30), "%s", tooltip "Control Mode", text variable: m_Instance.stat.sCtrlMode
    Rectangle (30,95 240x30), "%s", text variable: m_Instance.stat.sIDN
    Rectangle (30,120 240x30), "%s", text variable: m_Instance.stat.sRDI
    Button (65,300 150x60), "START"
        OnMouseClick: execute { m_bEnable := TRUE; }
    Button (65,370 150x60), "STOP"
        OnMouseClick: execute { m_bEnable := FALSE; }
    Lamp1 (680,407 25x25), tooltip "If ON, control output signal is active.", variable: m_Instance.q_bStart, style: Lamp-Lamp1-Green
    Rectangle (555,407 110x30), "Ctrl Signal :"
    Rectangle (457,242 246x30), "%s", tooltip "Control Mode", text variable: m_Instance.stat.sPumpState
END_VISUALIZATION

// ---- VISUs/Templates/GUI_TEMPLATE_CMD_OVERRIDE.TcVIS
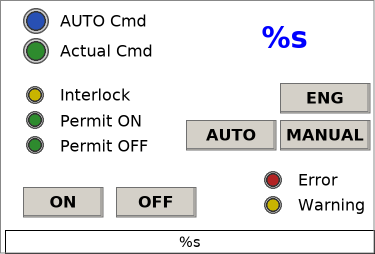
VISUALIZATION GUI_TEMPLATE_CMD_OVERRIDE  // 375x254
VAR_IN_OUT
	m_Cmd:		FB_CRYO_CMD_OVERRIDE;
END_VAR
    Lamp1 (25,85 20x20), variable: m_Cmd.out_bInterlock, style: Lamp-Lamp1-Yellow
    Lamp1 (25,110 20x20), variable: m_Cmd.bPermitOn, style: Lamp-Lamp1-Green
    Lamp1 (25,135 20x20), variable: m_Cmd.bPermitOff, style: Lamp-Lamp1-Green
    Rectangle (57,80 110x30), "Interlock"
    Rectangle (57,106 110x30), "Permit ON"
    Rectangle (57,131 110x30), "Permit OFF"
    Button (23,187 80x30), "ON", colour toggle: (m_Cmd.bPermitOn AND NOT m_Cmd.bAutoMode) OR m_Cmd.bEngMode, input disabled if: m_Cmd.bDisableBtnOn
        OnMouseClick: execute { m_Cmd.bManualCmd := TRUE; }
    Lamp1 (21,36 30x30), tooltip "Actual command going out", variable: m_Cmd.out_bEnable, style: Lamp-Lamp1-Green
    Rectangle (57,36 110x30), "Actual Cmd"
    Button (186,120 90x30), "AUTO", tooltip "Switch to AUTO Mode", colour toggle: m_Cmd.bAutoMode, input disabled if: m_Cmd.bAutoMode OR m_Cmd.bEngMode
        OnMouseClick: execute { m_Cmd.bAutoMode := TRUE; }
    Button (280,120 90x30), "MANUAL", tooltip "Switch to MANUAL Mode", colour toggle: NOT m_Cmd.bAutoMode, input disabled if: NOT m_Cmd.bAutoMode AND NOT m_Cmd.bEngMode
        OnMouseClick: execute { m_Cmd.bAutoMode := FALSE; }
    Button (116,187 80x30), "OFF", colour toggle: (m_Cmd.bPermitOff AND NOT m_Cmd.bAutoMode) OR m_Cmd.bEngMode, input disabled if: m_Cmd.bDisableBtnOff
        OnMouseClick: execute { m_Cmd.bManualCmd := FALSE; }
    Button (280,83 90x30), "ENG", tooltip "Toggle Engineering Mode", colour toggle: m_Cmd.bEngMode, input disabled if: m_Cmd.bAutoMode
        toggle m_Cmd.bEngMode
    Lamp1 (21,6 30x30), tooltip "Command coming from the Control System", variable: m_Cmd.in_bEnable, style: Lamp-Lamp1-Blue
    Rectangle (57,6 110x30), "AUTO Cmd"
    Rectangle (5,230 370x24), "%s", text variable: m_Cmd.out_sStatus
    Lamp1 (263,170 20x20), tooltip "If ON, there is an error in the SW implementation of permission handling.", variable: m_Cmd.out_bError, style: Lamp-Lamp1-Red
    Rectangle (295,165 75x30), "Error"
    Lamp1 (263,195 20x20), tooltip "If ON, ENG command is not safe!", variable: m_Cmd.out_bWarning, style: Lamp-Lamp1-Yellow
    Rectangle (295,190 75x30), "Warning"
    Rectangle (210,17 150x41), "%s", text variable: m_Cmd.out_sMode
END_VISUALIZATION

// ---- VISUs/Templates/GUI_TEMPLATE_CRYOTELGT.TcVIS
